LIN {X 0,Y 179.532,Z 337.35,A -85,B 0,C 180,E1 -23453.668,E2 -23453.668} C_VEL
LIN {X 0,Y 179.263,Z 347.509,A -85,B 0,C 180,E1 -23456.334,E2 -23456.334} C_VEL
LIN {X 0,Y 178.405,Z 355.039,A -85,B 0,C 180,E1 -23458.536,E2 -23458.536} C_VEL
LIN {X 0,Y 174.902,Z 363.864,A -85,B 0,C 180,E1 -23461.171,E2 -23461.171} C_VEL
LIN {X 0,Y 171.795,Z 371.251,A -85,B 0,C 180,E1 -23463.957,E2 -23463.957} C_VEL
LIN {X 0,Y 168.803,Z 378.338,A -85,B 0,C 180,E1 -23467.349,E2 -23467.349} C_VEL
LIN {X 0,Y 166.619,Z 383.189,A -85,B 0,C 180,E1 -23470.279,E2 -23470.279} C_VEL
LIN {X 0,Y 164.438,Z 387.902,A -85,B 0,C 180,E1 -23473.87,E2 -23473.87} C_VEL
LIN {X 0,Y 163.052,Z 391.511,A -85,B 0,C 180,E1 -23477.554,E2 -23477.554} C_VEL
LIN {X 0,Y 162.401,Z 393.372,A -85,B 0,C 180,E1 -23480.031,E2 -23480.031} C_VEL
LIN {X 0,Y 161.998,Z 394.77,A -85,B 0,C 180,E1 -23482.521,E2 -23482.521} C_VEL
LIN {X 0,Y 161.792,Z 395.77,A -85,B 0,C 180,E1 -23485.016,E2 -23485.016} C_VEL
LIN {X 0,Y 161.766,Z 396.433,A -85,B 0,C 180,E1 -23487.777,E2 -23487.777} C_VEL
LIN {X 0,Y 161.898,Z 396.597,A -85,B 0,C 180,E1 -23490,E2 -23490} C_VEL
LIN {X 0,Y 161.765,Z 396.367,A -85,B 0,C 180,E1 -23492.49,E2 -23492.49} C_VEL
LIN {X 0,Y 161.973,Z 394.738,A -85,B 0,C 180,E1 -23497.479,E2 -23497.479} C_VEL
LIN {X 0,Y 162.397,Z 393.327,A -85,B 0,C 180,E1 -23499.968,E2 -23499.968} C_VEL
LIN {X 0,Y 163.451,Z 390.371,A -85,B 0,C 180,E1 -23503.679,E2 -23503.679} C_VEL
LIN {X 0,Y 165.064,Z 386.378,A -85,B 0,C 180,E1 -23507.34,E2 -23507.34} C_VEL
LIN {X 0,Y 167.85,Z 380.247,A -85,B 0,C 180,E1 -23511.492,E2 -23511.492} C_VEL
LIN {X 0,Y 171.05,Z 373.162,A -85,B 0,C 180,E1 -23515.115,E2 -23515.115} C_VEL
LIN {X 0,Y 174.277,Z 365.256,A -85,B 0,C 180,E1 -23518.284,E2 -23518.284} C_VEL
LIN {X 0,Y 176.008,Z 361.044,A -85,B 0,C 180,E1 -23519.667,E2 -23519.667} C_VEL
LIN {X 0,Y 176.715,Z 358.334,A -85,B 0,C 180,E1 -23520.56,E2 -23520.56} C_VEL
LIN {X 0,Y 176.609,Z 354.361,A -85,B 0,C 180,E1 -23521.984,E2 -23521.984} C_VEL
LIN {X 0,Y 175.665,Z 350.503,A -85,B 0,C 180,E1 -23523.438,E2 -23523.438} C_VEL
LIN {X 0,Y 173.47,Z 342.313,A -85,B 0,C 180,E1 -23526.334,E2 -23526.334} C_VEL
LIN {X 0,Y 173.279,Z 339.26,A -85,B 0,C 180,E1 -23527.216,E2 -23527.216} C_VEL
LIN {X 0,Y 172.896,Z 328.815,A -85,B 0,C 180,E1 -23529.893,E2 -23529.893} C_VEL
LIN {X 0,Y 171.766,Z 319.398,A -85,B 0,C 180,E1 -23532.155,E2 -23532.155} C_VEL
LIN {X 0,Y 170.094,Z 313.723,A -85,B 0,C 180,E1 -23533.691,E2 -23533.691} C_VEL
LIN {X 0,Y 165.868,Z 303.988,A -85,B 0,C 180,E1 -23536.632,E2 -23536.632} C_VEL
LIN {X 0,Y 163.409,Z 299.193,A -85,B 0,C 180,E1 -23538.192,E2 -23538.192} C_VEL
LIN {X 0,Y 161.486,Z 295.384,A -85,B 0,C 180,E1 -23539.427,E2 -23539.427} C_VEL
LIN {X 0,Y 158.662,Z 290.982,A -85,B 0,C 180,E1 -23541.1,E2 -23541.1} C_VEL
LIN {X 0,Y 158.114,Z 289.125,A -85,B 0,C 180,E1 -23541.578,E2 -23541.578} C_VEL
LIN {X 0,Y 157.959,Z 287.633,A -85,B 0,C 180,E1 -23544.662,E2 -23544.662} C_VEL
LIN {X 0,Y 157.689,Z 286.213,A -85,B 0,C 180,E1 -23547.866,E2 -23547.866} C_VEL
LIN {X 0,Y 157.309,Z 283.978,A -85,B 0,C 180,E1 -23553.464,E2 -23553.464} C_VEL
LIN {X 0,Y 157.392,Z 283.88,A -85,B 0,C 180,E1 -23559.67,E2 -23559.67} C_VEL
LIN {X 0,Y 157.454,Z 283.87,A -85,B 0,C 180,E1 -23564.466,E2 -23564.466} C_VEL
LIN {X 0,Y 157.69,Z 283.841,A -85,B 0,C 180,E1 -23569.731,E2 -23569.731} C_VEL
LIN {X 0,Y 157.767,Z 283.83,A -85,B 0,C 180,E1 -23572.32,E2 -23572.32} C_VEL
LIN {X 0,Y 158.249,Z 283.773,A -85,B 0,C 180,E1 -23580,E2 -23580} C_VEL
LIN {X 0,Y 157.764,Z 283.832,A -85,B 0,C 180,E1 -23587.68,E2 -23587.68} C_VEL
LIN {X 0,Y 157.634,Z 283.847,A -85,B 0,C 180,E1 -23591.23,E2 -23591.23} C_VEL
LIN {X 0,Y 157.436,Z 283.871,A -85,B 0,C 180,E1 -23595.536,E2 -23595.536} C_VEL
LIN {X 0,Y 157.367,Z 283.88,A -85,B 0,C 180,E1 -23600.933,E2 -23600.933} C_VEL
LIN {X 0,Y 157.31,Z 283.888,A -85,B 0,C 180,E1 -23606.681,E2 -23606.681} C_VEL
LIN {X 0,Y 157.279,Z 283.895,A -85,B 0,C 180,E1 -23612.427,E2 -23612.427} C_VEL
LIN {X 0,Y 157.233,Z 283.899,A -85,B 0,C 180,E1 -23617.483,E2 -23617.483} C_VEL
LIN {X 0,Y 157.261,Z 284.165,A -85,B 0,C 180,E1 -23618.179,E2 -23618.179} C_VEL
LIN {X 0,Y 158.285,Z 286.868,A -85,B 0,C 180,E1 -23618.941,E2 -23618.941} C_VEL
LIN {X 0,Y 160.69,Z 289.727,A -85,B 0,C 180,E1 -23620.31,E2 -23620.31} C_VEL
LIN {X 0,Y 162.703,Z 293.411,A -85,B 0,C 180,E1 -23621.616,E2 -23621.616} C_VEL
LIN {X 0,Y 163.922,Z 295.532,A -85,B 0,C 180,E1 -23622.371,E2 -23622.371} C_VEL
LIN {X 0,Y 166.248,Z 299.878,A -85,B 0,C 180,E1 -23623.888,E2 -23623.888} C_VEL
LIN {X 0,Y 170.184,Z 308.553,A -85,B 0,C 180,E1 -23626.703,E2 -23626.703} C_VEL
LIN {X 0,Y 173.03,Z 318.057,A -85,B 0,C 180,E1 -23629.468,E2 -23629.468} C_VEL
LIN {X 0,Y 174.681,Z 328.982,A -85,B 0,C 180,E1 -23632.527,E2 -23632.527} C_VEL
LIN {X 0,Y 175.059,Z 338.675,A -85,B 0,C 180,E1 -23635.374,E2 -23635.374} C_VEL
LIN {X 0,Y 174.874,Z 343.244,A -85,B 0,C 180,E1 -23636.799,E2 -23636.799} C_VEL
LIN {X 0,Y 171.561,Z 351.776,A -85,B 0,C 180,E1 -23639.2,E2 -23639.2} C_VEL
LIN {X 0,Y 168.32,Z 359.639,A -85,B 0,C 180,E1 -23641.99,E2 -23641.99} C_VEL
LIN {X 0,Y 164.672,Z 367.301,A -85,B 0,C 180,E1 -23645.41,E2 -23645.41} C_VEL
LIN {X 0,Y 161.071,Z 374.352,A -85,B 0,C 180,E1 -23649.57,E2 -23649.57} C_VEL
LIN {X 0,Y 158.731,Z 379.04,A -85,B 0,C 180,E1 -23653.274,E2 -23653.274} C_VEL
LIN {X 0,Y 156.993,Z 382.624,A -85,B 0,C 180,E1 -23657.066,E2 -23657.066} C_VEL
LIN {X 0,Y 156.094,Z 384.475,A -85,B 0,C 180,E1 -23659.625,E2 -23659.625} C_VEL
LIN {X 0,Y 155.506,Z 385.863,A -85,B 0,C 180,E1 -23662.208,E2 -23662.208} C_VEL
LIN {X 0,Y 154.905,Z 387.455,A -85,B 0,C 180,E1 -23667.4,E2 -23667.4} C_VEL
LIN {X 0,Y 154.86,Z 387.681,A -85,B 0,C 180,E1 -23670,E2 -23670} C_VEL
LIN {X 0,Y 154.952,Z 387.273,A -85,B 0,C 180,E1 -23673.771,E2 -23673.771} C_VEL
LIN {X 0,Y 155.507,Z 385.933,A -85,B 0,C 180,E1 -23677.793,E2 -23677.793} C_VEL
LIN {X 0,Y 156.093,Z 384.576,A -85,B 0,C 180,E1 -23680.376,E2 -23680.376} C_VEL
LIN {X 0,Y 157.48,Z 381.707,A -85,B 0,C 180,E1 -23684.209,E2 -23684.209} C_VEL
LIN {X 0,Y 159.422,Z 377.814,A -85,B 0,C 180,E1 -23687.975,E2 -23687.975} C_VEL
LIN {X 0,Y 161.963,Z 372.79,A -85,B 0,C 180,E1 -23691.644,E2 -23691.644} C_VEL
LIN {X 0,Y 165.148,Z 366.457,A -85,B 0,C 180,E1 -23695.186,E2 -23695.186} C_VEL
LIN {X 0,Y 168.761,Z 358.637,A -85,B 0,C 180,E1 -23698.569,E2 -23698.569} C_VEL
LIN {X 0,Y 172.052,Z 350.641,A -85,B 0,C 180,E1 -23701.319,E2 -23701.319} C_VEL
LIN {X 0,Y 174.992,Z 342.742,A -85,B 0,C 180,E1 -23703.52,E2 -23703.52} C_VEL
LIN {X 0,Y 175.049,Z 333.244,A -85,B 0,C 180,E1 -23706.41,E2 -23706.41} C_VEL
LIN {X 0,Y 174.114,Z 324.129,A -85,B 0,C 180,E1 -23709.032,E2 -23709.032} C_VEL
LIN {X 0,Y 172.377,Z 315.457,A -85,B 0,C 180,E1 -23711.48,E2 -23711.48} C_VEL
LIN {X 0,Y 169.606,Z 307.081,A -85,B 0,C 180,E1 -23713.964,E2 -23713.964} C_VEL
LIN {X 0,Y 165.424,Z 298.191,A -85,B 0,C 180,E1 -23716.883,E2 -23716.883} C_VEL
LIN {X 0,Y 162.733,Z 293.422,A -85,B 0,C 180,E1 -23718.6,E2 -23718.6} C_VEL
LIN {X 0,Y 160.797,Z 289.973,A -85,B 0,C 180,E1 -23719.852,E2 -23719.852} C_VEL
LIN {X 0,Y 159.998,Z 288.814,A -85,B 0,C 180,E1 -23720.324,E2 -23720.324} C_VEL
LIN {X 0,Y 157.92,Z 286.258,A -85,B 0,C 180,E1 -23721.539,E2 -23721.539} C_VEL
LIN {X 0,Y 157.234,Z 283.938,A -85,B 0,C 180,E1 -23722.205,E2 -23722.205} C_VEL
LIN {X 0,Y 157.293,Z 283.894,A -85,B 0,C 180,E1 -23724.489,E2 -23724.489} C_VEL
LIN {X 0,Y 157.297,Z 283.889,A -85,B 0,C 180,E1 -23728.095,E2 -23728.095} C_VEL
LIN {X 0,Y 157.317,Z 283.885,A -85,B 0,C 180,E1 -23733.465,E2 -23733.465} C_VEL
LIN {X 0,Y 157.394,Z 283.878,A -85,B 0,C 180,E1 -23739.67,E2 -23739.67} C_VEL
LIN {X 0,Y 157.439,Z 283.874,A -85,B 0,C 180,E1 -23744.464,E2 -23744.464} C_VEL
LIN {X 0,Y 157.691,Z 283.842,A -85,B 0,C 180,E1 -23749.731,E2 -23749.731} C_VEL
LIN {X 0,Y 157.765,Z 283.834,A -85,B 0,C 180,E1 -23752.32,E2 -23752.32} C_VEL
LIN {X 0,Y 158.24,Z 283.773,A -85,B 0,C 180,E1 -23760,E2 -23760} C_VEL
LIN {X 0,Y 157.714,Z 283.838,A -85,B 0,C 180,E1 -23765.113,E2 -23765.113} C_VEL
LIN {X 0,Y 157.769,Z 283.83,A -85,B 0,C 180,E1 -23767.68,E2 -23767.68} C_VEL
LIN {X 0,Y 157.639,Z 283.849,A -85,B 0,C 180,E1 -23771.237,E2 -23771.237} C_VEL
LIN {X 0,Y 157.444,Z 283.872,A -85,B 0,C 180,E1 -23775.535,E2 -23775.535} C_VEL
LIN {X 0,Y 157.369,Z 283.882,A -85,B 0,C 180,E1 -23780.933,E2 -23780.933} C_VEL
LIN {X 0,Y 157.322,Z 284.102,A -85,B 0,C 180,E1 -23786.688,E2 -23786.688} C_VEL
LIN {X 0,Y 157.722,Z 286.361,A -85,B 0,C 180,E1 -23792.324,E2 -23792.324} C_VEL
LIN {X 0,Y 158.069,Z 288.406,A -85,B 0,C 180,E1 -23796.84,E2 -23796.84} C_VEL
LIN {X 0,Y 158.146,Z 289.255,A -85,B 0,C 180,E1 -23798.351,E2 -23798.351} C_VEL
LIN {X 0,Y 159.201,Z 292.065,A -85,B 0,C 180,E1 -23799.106,E2 -23799.106} C_VEL
LIN {X 0,Y 161.514,Z 295.42,A -85,B 0,C 180,E1 -23800.447,E2 -23800.447} C_VEL
LIN {X 0,Y 163.571,Z 299.367,A -85,B 0,C 180,E1 -23801.757,E2 -23801.757} C_VEL
LIN {X 0,Y 167.057,Z 306.433,A -85,B 0,C 180,E1 -23804.012,E2 -23804.012} C_VEL
LIN {X 0,Y 170.194,Z 313.991,A -85,B 0,C 180,E1 -23806.273,E2 -23806.273} C_VEL
LIN {X 0,Y 171.979,Z 320.43,A -85,B 0,C 180,E1 -23808.002,E2 -23808.002} C_VEL
LIN {X 0,Y 173.096,Z 330.614,A -85,B 0,C 180,E1 -23810.483,E2 -23810.483} C_VEL
LIN {X 0,Y 173.321,Z 341.13,A -85,B 0,C 180,E1 -23813.217,E2 -23813.217} C_VEL
LIN {X 0,Y 172.668,Z 350.737,A -85,B 0,C 180,E1 -23815.967,E2 -23815.967} C_VEL
LIN {X 0,Y 172.155,Z 354.834,A -85,B 0,C 180,E1 -23817.254,E2 -23817.254} C_VEL
LIN {X 0,Y 170.919,Z 358.58,A -85,B 0,C 180,E1 -23818.381,E2 -23818.381} C_VEL
LIN {X 0,Y 166.674,Z 368.22,A -85,B 0,C 180,E1 -23821.681,E2 -23821.681} C_VEL
LIN {X 0,Y 163.351,Z 375.904,A -85,B 0,C 180,E1 -23825.198,E2 -23825.198} C_VEL
LIN {X 0,Y 160.81,Z 381.168,A -85,B 0,C 180,E1 -23828.193,E2 -23828.193} C_VEL
LIN {X 0,Y 158.291,Z 386.268,A -85,B 0,C 180,E1 -23831.893,E2 -23831.893} C_VEL
LIN {X 0,Y 156.526,Z 390.236,A -85,B 0,C 180,E1 -23835.703,E2 -23835.703} C_VEL
LIN {X 0,Y 155.402,Z 393.173,A -85,B 0,C 180,E1 -23839.578,E2 -23839.578} C_VEL
LIN {X 0,Y 154.948,Z 394.57,A -85,B 0,C 180,E1 -23842.179,E2 -23842.179} C_VEL
LIN {X 0,Y 154.712,Z 395.57,A -85,B 0,C 180,E1 -23844.787,E2 -23844.787} C_VEL
LIN {X 0,Y 154.684,Z 396.297,A -85,B 0,C 180,E1 -23848.304,E2 -23848.304} C_VEL
LIN {X 0,Y 154.796,Z 396.397,A -85,B 0,C 180,E1 -23850,E2 -23850} C_VEL
LIN {X 0,Y 154.666,Z 396.167,A -85,B 0,C 180,E1 -23852.604,E2 -23852.604} C_VEL
LIN {X 0,Y 154.695,Z 395.547,A -85,B 0,C 180,E1 -23855.213,E2 -23855.213} C_VEL
LIN {X 0,Y 154.929,Z 394.538,A -85,B 0,C 180,E1 -23857.821,E2 -23857.821} C_VEL
LIN {X 0,Y 155.399,Z 393.126,A -85,B 0,C 180,E1 -23860.422,E2 -23860.422} C_VEL
LIN {X 0,Y 156.525,Z 390.17,A -85,B 0,C 180,E1 -23864.297,E2 -23864.297} C_VEL
LIN {X 0,Y 158.289,Z 386.177,A -85,B 0,C 180,E1 -23868.107,E2 -23868.107} C_VEL
LIN {X 0,Y 161.222,Z 380.045,A -85,B 0,C 180,E1 -23872.422,E2 -23872.422} C_VEL
LIN {X 0,Y 164.353,Z 373.538,A -85,B 0,C 180,E1 -23875.895,E2 -23875.895} C_VEL
LIN {X 0,Y 168.039,Z 365.054,A -85,B 0,C 180,E1 -23879.434,E2 -23879.434} C_VEL
LIN {X 0,Y 171.625,Z 356.544,A -85,B 0,C 180,E1 -23882.164,E2 -23882.164} C_VEL
LIN {X 0,Y 172.9,Z 348.293,A -85,B 0,C 180,E1 -23884.685,E2 -23884.685} C_VEL
LIN {X 0,Y 173.279,Z 339.26,A -85,B 0,C 180,E1 -23887.216,E2 -23887.216} C_VEL
LIN {X 0,Y 172.779,Z 334.847,A -85,B 0,C 180,E1 -23888.508,E2 -23888.508} C_VEL
LIN {X 0,Y 171.404,Z 330.8,A -85,B 0,C 180,E1 -23889.883,E2 -23889.883} C_VEL
LIN {X 0,Y 167.438,Z 323.176,A -85,B 0,C 180,E1 -23892.745,E2 -23892.745} C_VEL
LIN {X 0,Y 164.93,Z 317.767,A -85,B 0,C 180,E1 -23894.624,E2 -23894.624} C_VEL
LIN {X 0,Y 161.37,Z 308.826,A -85,B 0,C 180,E1 -23897.543,E2 -23897.543} C_VEL
LIN {X 0,Y 159.078,Z 304.056,A -85,B 0,C 180,E1 -23899.23,E2 -23899.23} C_VEL
LIN {X 0,Y 156.751,Z 299.454,A -85,B 0,C 180,E1 -23900.913,E2 -23900.913} C_VEL
LIN {X 0,Y 154.665,Z 295.601,A -85,B 0,C 180,E1 -23902.408,E2 -23902.408} C_VEL
LIN {X 0,Y 153.755,Z 294.127,A -85,B 0,C 180,E1 -23903.022,E2 -23903.022} C_VEL
LIN {X 0,Y 151.625,Z 290.908,A -85,B 0,C 180,E1 -23904.49,E2 -23904.49} C_VEL
LIN {X 0,Y 150.932,Z 288.787,A -85,B 0,C 180,E1 -23905.221,E2 -23905.221} C_VEL
LIN {X 0,Y 150.611,Z 287.176,A -85,B 0,C 180,E1 -23909.116,E2 -23909.116} C_VEL
LIN {X 0,Y 150.245,Z 284.971,A -85,B 0,C 180,E1 -23915.103,E2 -23915.103} C_VEL
LIN {X 0,Y 150.36,Z 284.757,A -85,B 0,C 180,E1 -23920.902,E2 -23920.902} C_VEL
LIN {X 0,Y 150.436,Z 284.743,A -85,B 0,C 180,E1 -23926.492,E2 -23926.492} C_VEL
LIN {X 0,Y 150.612,Z 284.721,A -85,B 0,C 180,E1 -23929.243,E2 -23929.243} C_VEL
LIN {X 0,Y 150.705,Z 284.709,A -85,B 0,C 180,E1 -23931.958,E2 -23931.958} C_VEL
LIN {X 0,Y 151.21,Z 284.65,A -85,B 0,C 180,E1 -23940,E2 -23940} C_VEL
LIN {X 0,Y 150.702,Z 284.71,A -85,B 0,C 180,E1 -23948.043,E2 -23948.043} C_VEL
LIN {X 0,Y 150.576,Z 284.725,A -85,B 0,C 180,E1 -23951.433,E2 -23951.433} C_VEL
LIN {X 0,Y 150.348,Z 284.756,A -85,B 0,C 180,E1 -23956.288,E2 -23956.288} C_VEL
LIN {X 0,Y 150.35,Z 284.755,A -85,B 0,C 180,E1 -23960.79,E2 -23960.79} C_VEL
LIN {X 0,Y 150.242,Z 284.769,A -85,B 0,C 180,E1 -23967.28,E2 -23967.28} C_VEL
LIN {X 0,Y 150.22,Z 284.774,A -85,B 0,C 180,E1 -23972.635,E2 -23972.635} C_VEL
LIN {X 0,Y 150.222,Z 284.912,A -85,B 0,C 180,E1 -23974.661,E2 -23974.661} C_VEL
LIN {X 0,Y 151.197,Z 287.513,A -85,B 0,C 180,E1 -23975.523,E2 -23975.523} C_VEL
LIN {X 0,Y 153.217,Z 289.733,A -85,B 0,C 180,E1 -23976.851,E2 -23976.851} C_VEL
LIN {X 0,Y 153.8,Z 290.482,A -85,B 0,C 180,E1 -23977.238,E2 -23977.238} C_VEL
LIN {X 0,Y 155.531,Z 293.516,A -85,B 0,C 180,E1 -23978.515,E2 -23978.515} C_VEL
LIN {X 0,Y 156.846,Z 295.277,A -85,B 0,C 180,E1 -23979.37,E2 -23979.37} C_VEL
LIN {X 0,Y 160.981,Z 303.073,A -85,B 0,C 180,E1 -23982.416,E2 -23982.416} C_VEL
LIN {X 0,Y 164.907,Z 312.263,A -85,B 0,C 180,E1 -23985.645,E2 -23985.645} C_VEL
LIN {X 0,Y 167.208,Z 320.482,A -85,B 0,C 180,E1 -23988.251,E2 -23988.251} C_VEL
LIN {X 0,Y 168.57,Z 330.571,A -85,B 0,C 180,E1 -23991.29,E2 -23991.29} C_VEL
LIN {X 0,Y 168.827,Z 339.162,A -85,B 0,C 180,E1 -23993.986,E2 -23993.986} C_VEL
LIN {X 0,Y 168.583,Z 344.502,A -85,B 0,C 180,E1 -23995.751,E2 -23995.751} C_VEL
LIN {X 0,Y 164.42,Z 354.389,A -85,B 0,C 180,E1 -23998.747,E2 -23998.747} C_VEL
LIN {X 0,Y 160.74,Z 362.559,A -85,B 0,C 180,E1 -24001.965,E2 -24001.965} C_VEL
LIN {X 0,Y 157.061,Z 369.724,A -85,B 0,C 180,E1 -24005.549,E2 -24005.549} C_VEL
LIN {X 0,Y 154.424,Z 374.553,A -85,B 0,C 180,E1 -24008.649,E2 -24008.649} C_VEL
LIN {X 0,Y 151.952,Z 379.241,A -85,B 0,C 180,E1 -24012.505,E2 -24012.505} C_VEL
LIN {X 0,Y 150.067,Z 382.825,A -85,B 0,C 180,E1 -24016.458,E2 -24016.458} C_VEL
LIN {X 0,Y 149.122,Z 384.675,A -85,B 0,C 180,E1 -24019.134,E2 -24019.134} C_VEL
LIN {X 0,Y 148.47,Z 386.063,A -85,B 0,C 180,E1 -24021.836,E2 -24021.836} C_VEL
LIN {X 0,Y 147.84,Z 387.549,A -85,B 0,C 180,E1 -24026.662,E2 -24026.662} C_VEL
LIN {X 0,Y 147.766,Z 387.881,A -85,B 0,C 180,E1 -24030,E2 -24030} C_VEL
LIN {X 0,Y 147.84,Z 387.579,A -85,B 0,C 180,E1 -24033.338,E2 -24033.338} C_VEL
LIN {X 0,Y 148.47,Z 386.133,A -85,B 0,C 180,E1 -24038.164,E2 -24038.164} C_VEL
LIN {X 0,Y 149.121,Z 384.775,A -85,B 0,C 180,E1 -24040.867,E2 -24040.867} C_VEL
LIN {X 0,Y 150.6,Z 381.906,A -85,B 0,C 180,E1 -24044.873,E2 -24044.873} C_VEL
LIN {X 0,Y 152.692,Z 378.012,A -85,B 0,C 180,E1 -24048.796,E2 -24048.796} C_VEL
LIN {X 0,Y 155.393,Z 372.988,A -85,B 0,C 180,E1 -24052.609,E2 -24052.609} C_VEL
LIN {X 0,Y 158.762,Z 366.655,A -85,B 0,C 180,E1 -24056.275,E2 -24056.275} C_VEL
LIN {X 0,Y 162.445,Z 359.077,A -85,B 0,C 180,E1 -24059.672,E2 -24059.672} C_VEL
LIN {X 0,Y 166.017,Z 350.839,A -85,B 0,C 180,E1 -24062.595,E2 -24062.595} C_VEL
LIN {X 0,Y 168.709,Z 344.004,A -85,B 0,C 180,E1 -24064.582,E2 -24064.582} C_VEL
LIN {X 0,Y 168.898,Z 334.156,A -85,B 0,C 180,E1 -24067.757,E2 -24067.757} C_VEL
LIN {X 0,Y 168.019,Z 325.162,A -85,B 0,C 180,E1 -24070.531,E2 -24070.531} C_VEL
LIN {X 0,Y 166.307,Z 316.8,A -85,B 0,C 180,E1 -24073.11,E2 -24073.11} C_VEL
LIN {X 0,Y 164.031,Z 309.92,A -85,B 0,C 180,E1 -24075.358,E2 -24075.358} C_VEL
LIN {X 0,Y 160.626,Z 302.512,A -85,B 0,C 180,E1 -24078.058,E2 -24078.058} C_VEL
LIN {X 0,Y 158.253,Z 298.012,A -85,B 0,C 180,E1 -24079.809,E2 -24079.809} C_VEL
LIN {X 0,Y 156.268,Z 294.386,A -85,B 0,C 180,E1 -24081.267,E2 -24081.267} C_VEL
LIN {X 0,Y 154.194,Z 291.412,A -85,B 0,C 180,E1 -24082.69,E2 -24082.69} C_VEL
LIN {X 0,Y 153.522,Z 289.91,A -85,B 0,C 180,E1 -24083.235,E2 -24083.235} C_VEL
LIN {X 0,Y 151.261,Z 287.635,A -85,B 0,C 180,E1 -24084.698,E2 -24084.698} C_VEL
LIN {X 0,Y 150.27,Z 285.206,A -85,B 0,C 180,E1 -24085.555,E2 -24085.555} C_VEL
LIN {X 0,Y 150.19,Z 284.773,A -85,B 0,C 180,E1 -24085.737,E2 -24085.737} C_VEL
LIN {X 0,Y 150.21,Z 284.769,A -85,B 0,C 180,E1 -24089.025,E2 -24089.025} C_VEL
LIN {X 0,Y 150.243,Z 284.763,A -85,B 0,C 180,E1 -24092.72,E2 -24092.72} C_VEL
LIN {X 0,Y 150.351,Z 284.757,A -85,B 0,C 180,E1 -24099.21,E2 -24099.21} C_VEL
LIN {X 0,Y 150.351,Z 284.758,A -85,B 0,C 180,E1 -24103.712,E2 -24103.712} C_VEL
LIN {X 0,Y 150.611,Z 284.725,A -85,B 0,C 180,E1 -24109.242,E2 -24109.242} C_VEL
LIN {X 0,Y 150.703,Z 284.713,A -85,B 0,C 180,E1 -24111.958,E2 -24111.958} C_VEL
LIN {X 0,Y 151.201,Z 284.65,A -85,B 0,C 180,E1 -24120,E2 -24120} C_VEL
LIN {X 0,Y 150.706,Z 284.711,A -85,B 0,C 180,E1 -24128.042,E2 -24128.042} C_VEL
LIN {X 0,Y 150.579,Z 284.729,A -85,B 0,C 180,E1 -24131.438,E2 -24131.438} C_VEL
LIN {X 0,Y 150.356,Z 284.757,A -85,B 0,C 180,E1 -24136.287,E2 -24136.287} C_VEL
LIN {X 0,Y 150.351,Z 284.757,A -85,B 0,C 180,E1 -24140.79,E2 -24140.79} C_VEL
LIN {X 0,Y 150.25,Z 285.039,A -85,B 0,C 180,E1 -24144.896,E2 -24144.896} C_VEL
LIN {X 0,Y 150.435,Z 286.08,A -85,B 0,C 180,E1 -24147.851,E2 -24147.851} C_VEL
LIN {X 0,Y 150.808,Z 288.09,A -85,B 0,C 180,E1 -24152.981,E2 -24152.981} C_VEL
LIN {X 0,Y 150.969,Z 288.997,A -85,B 0,C 180,E1 -24154.769,E2 -24154.769} C_VEL
LIN {X 0,Y 152.29,Z 292.195,A -85,B 0,C 180,E1 -24155.839,E2 -24155.839} C_VEL
LIN {X 0,Y 154.539,Z 295.267,A -85,B 0,C 180,E1 -24157.328,E2 -24157.328} C_VEL
LIN {X 0,Y 156.587,Z 299.181,A -85,B 0,C 180,E1 -24158.823,E2 -24158.823} C_VEL
LIN {X 0,Y 157.546,Z 300.81,A -85,B 0,C 180,E1 -24159.471,E2 -24159.471} C_VEL
LIN {X 0,Y 160.328,Z 306.492,A -85,B 0,C 180,E1 -24161.513,E2 -24161.513} C_VEL
LIN {X 0,Y 164.171,Z 315.549,A -85,B 0,C 180,E1 -24164.571,E2 -24164.571} C_VEL
LIN {X 0,Y 166.351,Z 322.936,A -85,B 0,C 180,E1 -24166.795,E2 -24166.795} C_VEL
LIN {X 0,Y 167.216,Z 333.484,A -85,B 0,C 180,E1 -24169.568,E2 -24169.568} C_VEL
LIN {X 0,Y 167.12,Z 343.551,A -85,B 0,C 180,E1 -24172.39,E2 -24172.39} C_VEL
LIN {X 0,Y 166.22,Z 352.654,A -85,B 0,C 180,E1 -24175.194,E2 -24175.194} C_VEL
LIN {X 0,Y 165.557,Z 356.585,A -85,B 0,C 180,E1 -24176.505,E2 -24176.505} C_VEL
LIN {X 0,Y 161.85,Z 365.045,A -85,B 0,C 180,E1 -24179.321,E2 -24179.321} C_VEL
LIN {X 0,Y 157.893,Z 373.389,A -85,B 0,C 180,E1 -24182.901,E2 -24182.901} C_VEL
LIN {X 0,Y 155.208,Z 378.961,A -85,B 0,C 180,E1 -24185.95,E2 -24185.95} C_VEL
LIN {X 0,Y 152.366,Z 384.481,A -85,B 0,C 180,E1 -24189.76,E2 -24189.76} C_VEL
LIN {X 0,Y 150.135,Z 388.812,A -85,B 0,C 180,E1 -24193.688,E2 -24193.688} C_VEL
LIN {X 0,Y 149.136,Z 391.111,A -85,B 0,C 180,E1 -24196.371,E2 -24196.371} C_VEL
LIN {X 0,Y 148.388,Z 392.973,A -85,B 0,C 180,E1 -24199.079,E2 -24199.079} C_VEL
LIN {X 0,Y 147.897,Z 394.37,A -85,B 0,C 180,E1 -24201.804,E2 -24201.804} C_VEL
LIN {X 0,Y 147.634,Z 395.37,A -85,B 0,C 180,E1 -24204.536,E2 -24204.536} C_VEL
LIN {X 0,Y 147.622,Z 396.131,A -85,B 0,C 180,E1 -24208.772,E2 -24208.772} C_VEL
LIN {X 0,Y 147.63,Z 396.118,A -85,B 0,C 180,E1 -24211.362,E2 -24211.362} C_VEL
LIN {X 0,Y 147.622,Z 395.346,A -85,B 0,C 180,E1 -24215.463,E2 -24215.463} C_VEL
LIN {X 0,Y 147.883,Z 394.337,A -85,B 0,C 180,E1 -24218.196,E2 -24218.196} C_VEL
LIN {X 0,Y 148.386,Z 392.925,A -85,B 0,C 180,E1 -24220.921,E2 -24220.921} C_VEL
LIN {X 0,Y 149.625,Z 389.968,A -85,B 0,C 180,E1 -24224.971,E2 -24224.971} C_VEL
LIN {X 0,Y 151.545,Z 385.975,A -85,B 0,C 180,E1 -24228.943,E2 -24228.943} C_VEL
LIN {X 0,Y 154.656,Z 379.843,A -85,B 0,C 180,E1 -24233.43,E2 -24233.43} C_VEL
LIN {X 0,Y 157.473,Z 374.39,A -85,B 0,C 180,E1 -24236.506,E2 -24236.506} C_VEL
LIN {X 0,Y 161.165,Z 366.342,A -85,B 0,C 180,E1 -24240.098,E2 -24240.098} C_VEL
LIN {X 0,Y 164.876,Z 358.148,A -85,B 0,C 180,E1 -24242.921,E2 -24242.921} C_VEL
LIN {X 0,Y 165.84,Z 354.367,A -85,B 0,C 180,E1 -24244.16,E2 -24244.16} C_VEL
LIN {X 0,Y 166.814,Z 346.89,A -85,B 0,C 180,E1 -24246.527,E2 -24246.527} C_VEL
LIN {X 0,Y 167.173,Z 336.191,A -85,B 0,C 180,E1 -24249.606,E2 -24249.606} C_VEL
LIN {X 0,Y 166.542,Z 325.417,A -85,B 0,C 180,E1 -24252.469,E2 -24252.469} C_VEL
LIN {X 0,Y 165.681,Z 320.289,A -85,B 0,C 180,E1 -24253.853,E2 -24253.853} C_VEL
LIN {X 0,Y 164.93,Z 317.767,A -85,B 0,C 180,E1 -24254.624,E2 -24254.624} C_VEL
LIN {X 0,Y 163.441,Z 315.395,A -85,B 0,C 180,E1 -24255.592,E2 -24255.592} C_VEL
LIN {X 0,Y 159.904,Z 312.847,A -85,B 0,C 180,E1 -24257.382,E2 -24257.382} C_VEL
LIN {X 0,Y 155.582,Z 309.957,A -85,B 0,C 180,E1 -24259.664,E2 -24259.664} C_VEL
LIN {X 0,Y 154.497,Z 308.525,A -85,B 0,C 180,E1 -24260.407,E2 -24260.407} C_VEL
LIN {X 0,Y 152.646,Z 304.534,A -85,B 0,C 180,E1 -24261.98,E2 -24261.98} C_VEL
LIN {X 0,Y 150.102,Z 299.628,A -85,B 0,C 180,E1 -24264.075,E2 -24264.075} C_VEL
LIN {X 0,Y 147.995,Z 295.975,A -85,B 0,C 180,E1 -24265.792,E2 -24265.792} C_VEL
LIN {X 0,Y 147.259,Z 294.473,A -85,B 0,C 180,E1 -24266.431,E2 -24266.431} C_VEL
LIN {X 0,Y 144.698,Z 291.323,A -85,B 0,C 180,E1 -24268.423,E2 -24268.423} C_VEL
LIN {X 0,Y 143.616,Z 288.48,A -85,B 0,C 180,E1 -24269.59,E2 -24269.59} C_VEL
LIN {X 0,Y 143.355,Z 286.976,A -85,B 0,C 180,E1 -24273.818,E2 -24273.818} C_VEL
LIN {X 0,Y 143.275,Z 285.64,A -85,B 0,C 180,E1 -24278.748,E2 -24278.748} C_VEL
LIN {X 0,Y 143.302,Z 285.635,A -85,B 0,C 180,E1 -24282.887,E2 -24282.887} C_VEL
LIN {X 0,Y 143.538,Z 285.603,A -85,B 0,C 180,E1 -24288.706,E2 -24288.706} C_VEL
LIN {X 0,Y 143.626,Z 285.592,A -85,B 0,C 180,E1 -24291.559,E2 -24291.559} C_VEL
LIN {X 0,Y 144.168,Z 285.527,A -85,B 0,C 180,E1 -24300,E2 -24300} C_VEL
LIN {X 0,Y 143.624,Z 285.591,A -85,B 0,C 180,E1 -24308.442,E2 -24308.442} C_VEL
LIN {X 0,Y 143.502,Z 285.606,A -85,B 0,C 180,E1 -24311.623,E2 -24311.623} C_VEL
LIN {X 0,Y 143.292,Z 285.636,A -85,B 0,C 180,E1 -24317.115,E2 -24317.115} C_VEL
LIN {X 0,Y 143.275,Z 285.635,A -85,B 0,C 180,E1 -24321.252,E2 -24321.252} C_VEL
LIN {X 0,Y 143.189,Z 285.65,A -85,B 0,C 180,E1 -24327.936,E2 -24327.936} C_VEL
LIN {X 0,Y 143.171,Z 285.824,A -85,B 0,C 180,E1 -24330.413,E2 -24330.413} C_VEL
LIN {X 0,Y 144.091,Z 288.37,A -85,B 0,C 180,E1 -24331.418,E2 -24331.418} C_VEL
LIN {X 0,Y 146.142,Z 290.577,A -85,B 0,C 180,E1 -24333.039,E2 -24333.039} C_VEL
LIN {X 0,Y 147.053,Z 291.396,A -85,B 0,C 180,E1 -24333.72,E2 -24333.72} C_VEL
LIN {X 0,Y 148.8,Z 294.569,A -85,B 0,C 180,E1 -24335.247,E2 -24335.247} C_VEL
LIN {X 0,Y 150.25,Z 296.219,A -85,B 0,C 180,E1 -24336.3,E2 -24336.3} C_VEL
LIN {X 0,Y 152.147,Z 299.508,A -85,B 0,C 180,E1 -24337.868,E2 -24337.868} C_VEL
LIN {X 0,Y 156.248,Z 307.471,A -85,B 0,C 180,E1 -24341.311,E2 -24341.311} C_VEL
LIN {X 0,Y 159.781,Z 316.43,A -85,B 0,C 180,E1 -24344.73,E2 -24344.73} C_VEL
LIN {X 0,Y 161.779,Z 324.81,A -85,B 0,C 180,E1 -24347.605,E2 -24347.605} C_VEL
LIN {X 0,Y 162.726,Z 335.269,A -85,B 0,C 180,E1 -24351.024,E2 -24351.024} C_VEL
LIN {X 0,Y 162.393,Z 344.718,A -85,B 0,C 180,E1 -24354.25,E2 -24354.25} C_VEL
LIN {X 0,Y 161.922,Z 346.659,A -85,B 0,C 180,E1 -24354.894,E2 -24354.894} C_VEL
LIN {X 0,Y 157.969,Z 355.485,A -85,B 0,C 180,E1 -24357.732,E2 -24357.732} C_VEL
LIN {X 0,Y 154.498,Z 362.761,A -85,B 0,C 180,E1 -24360.725,E2 -24360.725} C_VEL
LIN {X 0,Y 150.641,Z 369.925,A -85,B 0,C 180,E1 -24364.434,E2 -24364.434} C_VEL
LIN {X 0,Y 147.822,Z 374.755,A -85,B 0,C 180,E1 -24367.645,E2 -24367.645} C_VEL
LIN {X 0,Y 145.187,Z 379.442,A -85,B 0,C 180,E1 -24371.661,E2 -24371.661} C_VEL
LIN {X 0,Y 143.171,Z 383.026,A -85,B 0,C 180,E1 -24375.792,E2 -24375.792} C_VEL
LIN {X 0,Y 142.149,Z 384.876,A -85,B 0,C 180,E1 -24378.594,E2 -24378.594} C_VEL
LIN {X 0,Y 141.435,Z 386.264,A -85,B 0,C 180,E1 -24381.427,E2 -24381.427} C_VEL
LIN {X 0,Y 141.007,Z 387.249,A -85,B 0,C 180,E1 -24384.279,E2 -24384.279} C_VEL
LIN {X 0,Y 140.736,Z 387.855,A -85,B 0,C 180,E1 -24387.138,E2 -24387.138} C_VEL
LIN {X 0,Y 140.69,Z 388.08,A -85,B 0,C 180,E1 -24390,E2 -24390} C_VEL
LIN {X 0,Y 140.737,Z 387.885,A -85,B 0,C 180,E1 -24392.863,E2 -24392.863} C_VEL
LIN {X 0,Y 141.007,Z 387.298,A -85,B 0,C 180,E1 -24395.721,E2 -24395.721} C_VEL
LIN {X 0,Y 142.148,Z 384.975,A -85,B 0,C 180,E1 -24401.407,E2 -24401.407} C_VEL
LIN {X 0,Y 143.751,Z 382.105,A -85,B 0,C 180,E1 -24405.599,E2 -24405.599} C_VEL
LIN {X 0,Y 145.975,Z 378.212,A -85,B 0,C 180,E1 -24409.696,E2 -24409.696} C_VEL
LIN {X 0,Y 148.848,Z 373.187,A -85,B 0,C 180,E1 -24413.662,E2 -24413.662} C_VEL
LIN {X 0,Y 152.44,Z 366.852,A -85,B 0,C 180,E1 -24417.454,E2 -24417.454} C_VEL
LIN {X 0,Y 156.196,Z 359.52,A -85,B 0,C 180,E1 -24420.862,E2 -24420.862} C_VEL
LIN {X 0,Y 160.153,Z 350.86,A -85,B 0,C 180,E1 -24424.021,E2 -24424.021} C_VEL
LIN {X 0,Y 162.458,Z 345.218,A -85,B 0,C 180,E1 -24425.734,E2 -24425.734} C_VEL
LIN {X 0,Y 162.837,Z 335.654,A -85,B 0,C 180,E1 -24429.024,E2 -24429.024} C_VEL
LIN {X 0,Y 162.115,Z 326.992,A -85,B 0,C 180,E1 -24431.894,E2 -24431.894} C_VEL
LIN {X 0,Y 160.636,Z 319.408,A -85,B 0,C 180,E1 -24434.429,E2 -24434.429} C_VEL
LIN {X 0,Y 158.121,Z 311.712,A -85,B 0,C 180,E1 -24437.237,E2 -24437.237} C_VEL
LIN {X 0,Y 154.49,Z 303.853,A -85,B 0,C 180,E1 -24440.44,E2 -24440.44} C_VEL
LIN {X 0,Y 152.235,Z 299.664,A -85,B 0,C 180,E1 -24442.319,E2 -24442.319} C_VEL
LIN {X 0,Y 150.214,Z 296.148,A -85,B 0,C 180,E1 -24444.002,E2 -24444.002} C_VEL
LIN {X 0,Y 147.506,Z 292.542,A -85,B 0,C 180,E1 -24446.106,E2 -24446.106} C_VEL
LIN {X 0,Y 146.77,Z 290.978,A -85,B 0,C 180,E1 -24446.81,E2 -24446.81} C_VEL
LIN {X 0,Y 144.458,Z 288.915,A -85,B 0,C 180,E1 -24448.568,E2 -24448.568} C_VEL
LIN {X 0,Y 143.292,Z 286.509,A -85,B 0,C 180,E1 -24449.717,E2 -24449.717} C_VEL
LIN {X 0,Y 143.137,Z 285.652,A -85,B 0,C 180,E1 -24449.986,E2 -24449.986} C_VEL
LIN {X 0,Y 143.157,Z 285.65,A -85,B 0,C 180,E1 -24453.779,E2 -24453.779} C_VEL
LIN {X 0,Y 143.307,Z 285.632,A -85,B 0,C 180,E1 -24459.922,E2 -24459.922} C_VEL
LIN {X 0,Y 143.326,Z 285.631,A -85,B 0,C 180,E1 -24465.808,E2 -24465.808} C_VEL
LIN {X 0,Y 143.537,Z 285.604,A -85,B 0,C 180,E1 -24468.705,E2 -24468.705} C_VEL
LIN {X 0,Y 143.625,Z 285.594,A -85,B 0,C 180,E1 -24471.558,E2 -24471.558} C_VEL
LIN {X 0,Y 144.159,Z 285.527,A -85,B 0,C 180,E1 -24480,E2 -24480} C_VEL
LIN {X 0,Y 143.628,Z 285.594,A -85,B 0,C 180,E1 -24488.441,E2 -24488.441} C_VEL
LIN {X 0,Y 143.507,Z 285.61,A -85,B 0,C 180,E1 -24491.629,E2 -24491.629} C_VEL
LIN {X 0,Y 143.298,Z 285.633,A -85,B 0,C 180,E1 -24497.114,E2 -24497.114} C_VEL
LIN {X 0,Y 143.276,Z 285.637,A -85,B 0,C 180,E1 -24501.252,E2 -24501.252} C_VEL
LIN {X 0,Y 143.505,Z 287.728,A -85,B 0,C 180,E1 -24508.172,E2 -24508.172} C_VEL
LIN {X 0,Y 143.647,Z 288.601,A -85,B 0,C 180,E1 -24510.301,E2 -24510.301} C_VEL
LIN {X 0,Y 144.981,Z 291.774,A -85,B 0,C 180,E1 -24511.61,E2 -24511.61} C_VEL
LIN {X 0,Y 147.678,Z 295.066,A -85,B 0,C 180,E1 -24513.698,E2 -24513.698} C_VEL
LIN {X 0,Y 149.466,Z 298.742,A -85,B 0,C 180,E1 -24515.273,E2 -24515.273} C_VEL
LIN {X 0,Y 150.856,Z 300.912,A -85,B 0,C 180,E1 -24516.337,E2 -24516.337} C_VEL
LIN {X 0,Y 153.336,Z 305.758,A -85,B 0,C 180,E1 -24518.393,E2 -24518.393} C_VEL
LIN {X 0,Y 156.791,Z 313.489,A -85,B 0,C 180,E1 -24521.388,E2 -24521.388} C_VEL
LIN {X 0,Y 159.672,Z 321.484,A -85,B 0,C 180,E1 -24524.232,E2 -24524.232} C_VEL
LIN {X 0,Y 160.698,Z 325.686,A -85,B 0,C 180,E1 -24525.593,E2 -24525.593} C_VEL
LIN {X 0,Y 161.274,Z 335.349,A -85,B 0,C 180,E1 -24528.344,E2 -24528.344} C_VEL
LIN {X 0,Y 160.903,Z 345.837,A -85,B 0,C 180,E1 -24531.508,E2 -24531.508} C_VEL
LIN {X 0,Y 159.794,Z 354.42,A -85,B 0,C 180,E1 -24534.355,E2 -24534.355} C_VEL
LIN {X 0,Y 158.909,Z 358.183,A -85,B 0,C 180,E1 -24535.675,E2 -24535.675} C_VEL
LIN {X 0,Y 154.285,Z 367.824,A -85,B 0,C 180,E1 -24539.172,E2 -24539.172} C_VEL
LIN {X 0,Y 150.467,Z 375.504,A -85,B 0,C 180,E1 -24542.909,E2 -24542.909} C_VEL
LIN {X 0,Y 146.647,Z 382.59,A -85,B 0,C 180,E1 -24547.455,E2 -24547.455} C_VEL
LIN {X 0,Y 144.025,Z 387.304,A -85,B 0,C 180,E1 -24551.507,E2 -24551.507} C_VEL
LIN {X 0,Y 142.219,Z 390.911,A -85,B 0,C 180,E1 -24555.695,E2 -24555.695} C_VEL
LIN {X 0,Y 141.399,Z 392.773,A -85,B 0,C 180,E1 -24558.532,E2 -24558.532} C_VEL
LIN {X 0,Y 140.848,Z 394.17,A -85,B 0,C 180,E1 -24561.391,E2 -24561.391} C_VEL
LIN {X 0,Y 140.555,Z 395.171,A -85,B 0,C 180,E1 -24564.26,E2 -24564.26} C_VEL
LIN {X 0,Y 140.569,Z 395.969,A -85,B 0,C 180,E1 -24569.356,E2 -24569.356} C_VEL
LIN {X 0,Y 140.486,Z 395.767,A -85,B 0,C 180,E1 -24572.867,E2 -24572.867} C_VEL
LIN {X 0,Y 140.545,Z 395.146,A -85,B 0,C 180,E1 -24575.74,E2 -24575.74} C_VEL
LIN {X 0,Y 140.837,Z 394.136,A -85,B 0,C 180,E1 -24578.61,E2 -24578.61} C_VEL
LIN {X 0,Y 141.397,Z 392.724,A -85,B 0,C 180,E1 -24581.467,E2 -24581.467} C_VEL
LIN {X 0,Y 142.727,Z 389.766,A -85,B 0,C 180,E1 -24585.713,E2 -24585.713} C_VEL
LIN {X 0,Y 144.81,Z 385.773,A -85,B 0,C 180,E1 -24589.86,E2 -24589.86} C_VEL
LIN {X 0,Y 148.154,Z 379.641,A -85,B 0,C 180,E1 -24594.524,E2 -24594.524} C_VEL
LIN {X 0,Y 151.556,Z 373.198,A -85,B 0,C 180,E1 -24598.227,E2 -24598.227} C_VEL
LIN {X 0,Y 155.789,Z 364.648,A -85,B 0,C 180,E1 -24602.01,E2 -24602.01} C_VEL
LIN {X 0,Y 158.871,Z 357.942,A -85,B 0,C 180,E1 -24604.334,E2 -24604.334} C_VEL
LIN {X 0,Y 160.325,Z 350.607,A -85,B 0,C 180,E1 -24606.856,E2 -24606.856} C_VEL
LIN {X 0,Y 161.123,Z 340.524,A -85,B 0,C 180,E1 -24610.043,E2 -24610.043} C_VEL
LIN {X 0,Y 161.008,Z 330.267,A -85,B 0,C 180,E1 -24613.019,E2 -24613.019} C_VEL
LIN {X 0,Y 160.554,Z 325.178,A -85,B 0,C 180,E1 -24614.457,E2 -24614.457} C_VEL
LIN {X 0,Y 158.621,Z 318.437,A -85,B 0,C 180,E1 -24616.713,E2 -24616.713} C_VEL
LIN {X 0,Y 155.251,Z 309.829,A -85,B 0,C 180,E1 -24619.829,E2 -24619.829} C_VEL
LIN {X 0,Y 154.497,Z 308.525,A -85,B 0,C 180,E1 -24620.407,E2 -24620.407} C_VEL
LIN {X 0,Y 152.771,Z 306.643,A -85,B 0,C 180,E1 -24621.557,E2 -24621.557} C_VEL
LIN {X 0,Y 145.769,Z 303.209,A -85,B 0,C 180,E1 -24625.795,E2 -24625.795} C_VEL
LIN {X 0,Y 144.348,Z 301.181,A -85,B 0,C 180,E1 -24627.02,E2 -24627.02} C_VEL
LIN {X 0,Y 143.478,Z 299.794,A -85,B 0,C 180,E1 -24627.812,E2 -24627.812} C_VEL
LIN {X 0,Y 141.291,Z 296.443,A -85,B 0,C 180,E1 -24629.863,E2 -24629.863} C_VEL
LIN {X 0,Y 140.388,Z 294.444,A -85,B 0,C 180,E1 -24630.868,E2 -24630.868} C_VEL
LIN {X 0,Y 137.602,Z 291.237,A -85,B 0,C 180,E1 -24633.557,E2 -24633.557} C_VEL
LIN {X 0,Y 136.422,Z 288.447,A -85,B 0,C 180,E1 -24635.052,E2 -24635.052} C_VEL
LIN {X 0,Y 136.315,Z 288.076,A -85,B 0,C 180,E1 -24635.235,E2 -24635.235} C_VEL
LIN {X 0,Y 136.305,Z 286.985,A -85,B 0,C 180,E1 -24638.843,E2 -24638.843} C_VEL
LIN {X 0,Y 136.242,Z 286.513,A -85,B 0,C 180,E1 -24641.97,E2 -24641.97} C_VEL
LIN {X 0,Y 136.445,Z 286.489,A -85,B 0,C 180,E1 -24648.138,E2 -24648.138} C_VEL
LIN {X 0,Y 136.552,Z 286.475,A -85,B 0,C 180,E1 -24651.118,E2 -24651.118} C_VEL
LIN {X 0,Y 137.125,Z 286.405,A -85,B 0,C 180,E1 -24660,E2 -24660} C_VEL
LIN {X 0,Y 136.55,Z 286.472,A -85,B 0,C 180,E1 -24668.882,E2 -24668.882} C_VEL
LIN {X 0,Y 136.418,Z 286.488,A -85,B 0,C 180,E1 -24671.892,E2 -24671.892} C_VEL
LIN {X 0,Y 136.21,Z 286.515,A -85,B 0,C 180,E1 -24678.034,E2 -24678.034} C_VEL
LIN {X 0,Y 136.197,Z 286.517,A -85,B 0,C 180,E1 -24681.746,E2 -24681.746} C_VEL
LIN {X 0,Y 136.082,Z 286.55,A -85,B 0,C 180,E1 -24684.913,E2 -24684.913} C_VEL
LIN {X 0,Y 136.877,Z 288.957,A -85,B 0,C 180,E1 -24686.081,E2 -24686.081} C_VEL
LIN {X 0,Y 139.007,Z 291.406,A -85,B 0,C 180,E1 -24688.276,E2 -24688.276} C_VEL
LIN {X 0,Y 140.257,Z 292.337,A -85,B 0,C 180,E1 -24689.413,E2 -24689.413} C_VEL
LIN {X 0,Y 141.843,Z 295.435,A -85,B 0,C 180,E1 -24691.142,E2 -24691.142} C_VEL
LIN {X 0,Y 143.796,Z 297.482,A -85,B 0,C 180,E1 -24692.834,E2 -24692.834} C_VEL
LIN {X 0,Y 145.757,Z 300.869,A -85,B 0,C 180,E1 -24694.72,E2 -24694.72} C_VEL
LIN {X 0,Y 146.541,Z 301.901,A -85,B 0,C 180,E1 -24695.383,E2 -24695.383} C_VEL
LIN {X 0,Y 150.035,Z 308.663,A -85,B 0,C 180,E1 -24698.753,E2 -24698.753} C_VEL
LIN {X 0,Y 152.93,Z 315.579,A -85,B 0,C 180,E1 -24701.789,E2 -24701.789} C_VEL
LIN {X 0,Y 155.145,Z 322.61,A -85,B 0,C 180,E1 -24704.6,E2 -24704.6} C_VEL
LIN {X 0,Y 156.251,Z 329.097,A -85,B 0,C 180,E1 -24706.963,E2 -24706.963} C_VEL
LIN {X 0,Y 156.686,Z 338.746,A -85,B 0,C 180,E1 -24710.38,E2 -24710.38} C_VEL
LIN {X 0,Y 156.032,Z 346.867,A -85,B 0,C 180,E1 -24713.358,E2 -24713.358} C_VEL
LIN {X 0,Y 151.887,Z 355.94,A -85,B 0,C 180,E1 -24716.396,E2 -24716.396} C_VEL
LIN {X 0,Y 147.653,Z 364.288,A -85,B 0,C 180,E1 -24720.015,E2 -24720.015} C_VEL
LIN {X 0,Y 143.642,Z 371.151,A -85,B 0,C 180,E1 -24723.874,E2 -24723.874} C_VEL
LIN {X 0,Y 140.288,Z 376.644,A -85,B 0,C 180,E1 -24727.931,E2 -24727.931} C_VEL
LIN {X 0,Y 137.67,Z 380.95,A -85,B 0,C 180,E1 -24732.164,E2 -24732.164} C_VEL
LIN {X 0,Y 136.306,Z 383.226,A -85,B 0,C 180,E1 -24735.061,E2 -24735.061} C_VEL
LIN {X 0,Y 135.185,Z 385.077,A -85,B 0,C 180,E1 -24737.998,E2 -24737.998} C_VEL
LIN {X 0,Y 134.429,Z 386.464,A -85,B 0,C 180,E1 -24740.977,E2 -24740.977} C_VEL
LIN {X 0,Y 133.949,Z 387.449,A -85,B 0,C 180,E1 -24743.977,E2 -24743.977} C_VEL
LIN {X 0,Y 133.579,Z 388.204,A -85,B 0,C 180,E1 -24748.494,E2 -24748.494} C_VEL
LIN {X 0,Y 133.659,Z 388.084,A -85,B 0,C 180,E1 -24753.014,E2 -24753.014} C_VEL
LIN {X 0,Y 133.949,Z 387.498,A -85,B 0,C 180,E1 -24756.024,E2 -24756.024} C_VEL
LIN {X 0,Y 135.183,Z 385.174,A -85,B 0,C 180,E1 -24762.003,E2 -24762.003} C_VEL
LIN {X 0,Y 136.917,Z 382.304,A -85,B 0,C 180,E1 -24766.399,E2 -24766.399} C_VEL
LIN {X 0,Y 139.303,Z 378.41,A -85,B 0,C 180,E1 -24770.681,E2 -24770.681} C_VEL
LIN {X 0,Y 142.364,Z 373.386,A -85,B 0,C 180,E1 -24774.811,E2 -24774.811} C_VEL
LIN {X 0,Y 146.174,Z 367.05,A -85,B 0,C 180,E1 -24778.738,E2 -24778.738} C_VEL
LIN {X 0,Y 149.89,Z 360.212,A -85,B 0,C 180,E1 -24782.048,E2 -24782.048} C_VEL
LIN {X 0,Y 154.333,Z 351.055,A -85,B 0,C 180,E1 -24785.494,E2 -24785.494} C_VEL
LIN {X 0,Y 156.022,Z 347.353,A -85,B 0,C 180,E1 -24786.645,E2 -24786.645} C_VEL
LIN {X 0,Y 156.734,Z 340.126,A -85,B 0,C 180,E1 -24789.318,E2 -24789.318} C_VEL
LIN {X 0,Y 156.52,Z 331.701,A -85,B 0,C 180,E1 -24792.34,E2 -24792.34} C_VEL
LIN {X 0,Y 155.469,Z 324.094,A -85,B 0,C 180,E1 -24795.064,E2 -24795.064} C_VEL
LIN {X 0,Y 153.699,Z 317.643,A -85,B 0,C 180,E1 -24797.588,E2 -24797.588} C_VEL
LIN {X 0,Y 150.606,Z 309.891,A -85,B 0,C 180,E1 -24800.935,E2 -24800.935} C_VEL
LIN {X 0,Y 148.566,Z 305.496,A -85,B 0,C 180,E1 -24802.989,E2 -24802.989} C_VEL
LIN {X 0,Y 146.579,Z 301.914,A -85,B 0,C 180,E1 -24804.875,E2 -24804.875} C_VEL
LIN {X 0,Y 143.854,Z 297.682,A -85,B 0,C 180,E1 -24807.389,E2 -24807.389} C_VEL
LIN {X 0,Y 143.054,Z 296.68,A -85,B 0,C 180,E1 -24808.121,E2 -24808.121} C_VEL
LIN {X 0,Y 140.945,Z 293.978,A -85,B 0,C 180,E1 -24810.09,E2 -24810.09} C_VEL
LIN {X 0,Y 140.174,Z 292.087,A -85,B 0,C 180,E1 -24811.036,E2 -24811.036} C_VEL
LIN {X 0,Y 137.615,Z 290.057,A -85,B 0,C 180,E1 -24813.457,E2 -24813.457} C_VEL
LIN {X 0,Y 136.265,Z 287.508,A -85,B 0,C 180,E1 -24815.123,E2 -24815.123} C_VEL
LIN {X 0,Y 136.083,Z 286.528,A -85,B 0,C 180,E1 -24815.596,E2 -24815.596} C_VEL
LIN {X 0,Y 136.244,Z 286.515,A -85,B 0,C 180,E1 -24818.833,E2 -24818.833} C_VEL
LIN {X 0,Y 136.247,Z 286.511,A -85,B 0,C 180,E1 -24825.053,E2 -24825.053} C_VEL
LIN {X 0,Y 136.427,Z 286.489,A -85,B 0,C 180,E1 -24828.177,E2 -24828.177} C_VEL
LIN {X 0,Y 136.55,Z 286.474,A -85,B 0,C 180,E1 -24831.118,E2 -24831.118} C_VEL
LIN {X 0,Y 137.116,Z 286.404,A -85,B 0,C 180,E1 -24840,E2 -24840} C_VEL
LIN {X 0,Y 136.553,Z 286.476,A -85,B 0,C 180,E1 -24848.882,E2 -24848.882} C_VEL
LIN {X 0,Y 136.442,Z 286.488,A -85,B 0,C 180,E1 -24851.89,E2 -24851.89} C_VEL
LIN {X 0,Y 136.24,Z 286.514,A -85,B 0,C 180,E1 -24858.03,E2 -24858.03} C_VEL
LIN {X 0,Y 136.306,Z 287.256,A -85,B 0,C 180,E1 -24861.86,E2 -24861.86} C_VEL
LIN {X 0,Y 136.354,Z 288.192,A -85,B 0,C 180,E1 -24864.554,E2 -24864.554} C_VEL
LIN {X 0,Y 137.434,Z 290.903,A -85,B 0,C 180,E1 -24865.968,E2 -24865.968} C_VEL
LIN {X 0,Y 139.983,Z 294.053,A -85,B 0,C 180,E1 -24868.529,E2 -24868.529} C_VEL
LIN {X 0,Y 140.788,Z 295.024,A -85,B 0,C 180,E1 -24869.28,E2 -24869.28} C_VEL
LIN {X 0,Y 142.556,Z 298.639,A -85,B 0,C 180,E1 -24871.175,E2 -24871.175} C_VEL
LIN {X 0,Y 144.217,Z 300.811,A -85,B 0,C 180,E1 -24872.622,E2 -24872.622} C_VEL
LIN {X 0,Y 146.302,Z 304.971,A -85,B 0,C 180,E1 -24874.677,E2 -24874.677} C_VEL
LIN {X 0,Y 149.399,Z 311.633,A -85,B 0,C 180,E1 -24877.701,E2 -24877.701} C_VEL
LIN {X 0,Y 151.986,Z 317.895,A -85,B 0,C 180,E1 -24880.344,E2 -24880.344} C_VEL
LIN {X 0,Y 154.754,Z 326.771,A -85,B 0,C 180,E1 -24883.742,E2 -24883.742} C_VEL
LIN {X 0,Y 155.361,Z 332.01,A -85,B 0,C 180,E1 -24885.436,E2 -24885.436} C_VEL
LIN {X 0,Y 155.251,Z 341.976,A -85,B 0,C 180,E1 -24888.543,E2 -24888.543} C_VEL
LIN {X 0,Y 154.229,Z 351.449,A -85,B 0,C 180,E1 -24891.718,E2 -24891.718} C_VEL
LIN {X 0,Y 152.946,Z 357.98,A -85,B 0,C 180,E1 -24894.135,E2 -24894.135} C_VEL
LIN {X 0,Y 148.987,Z 366.139,A -85,B 0,C 180,E1 -24897.147,E2 -24897.147} C_VEL
LIN {X 0,Y 144.716,Z 374.148,A -85,B 0,C 180,E1 -24900.945,E2 -24900.945} C_VEL
LIN {X 0,Y 141.72,Z 379.576,A -85,B 0,C 180,E1 -24904.283,E2 -24904.283} C_VEL
LIN {X 0,Y 138.127,Z 385.67,A -85,B 0,C 180,E1 -24909.135,E2 -24909.135} C_VEL
LIN {X 0,Y 135.868,Z 389.636,A -85,B 0,C 180,E1 -24913.471,E2 -24913.471} C_VEL
LIN {X 0,Y 134.434,Z 392.573,A -85,B 0,C 180,E1 -24917.929,E2 -24917.929} C_VEL
LIN {X 0,Y 133.822,Z 393.971,A -85,B 0,C 180,E1 -24920.935,E2 -24920.935} C_VEL
LIN {X 0,Y 133.398,Z 395.583,A -85,B 0,C 180,E1 -24926.98,E2 -24926.98} C_VEL
LIN {X 0,Y 133.532,Z 395.798,A -85,B 0,C 180,E1 -24930,E2 -24930} C_VEL
LIN {X 0,Y 133.397,Z 395.567,A -85,B 0,C 180,E1 -24933.02,E2 -24933.02} C_VEL
LIN {X 0,Y 133.814,Z 393.936,A -85,B 0,C 180,E1 -24939.065,E2 -24939.065} C_VEL
LIN {X 0,Y 134.432,Z 392.523,A -85,B 0,C 180,E1 -24942.07,E2 -24942.07} C_VEL
LIN {X 0,Y 135.867,Z 389.564,A -85,B 0,C 180,E1 -24946.529,E2 -24946.529} C_VEL
LIN {X 0,Y 138.124,Z 385.572,A -85,B 0,C 180,E1 -24950.865,E2 -24950.865} C_VEL
LIN {X 0,Y 141.718,Z 379.439,A -85,B 0,C 180,E1 -24955.717,E2 -24955.717} C_VEL
LIN {X 0,Y 145.366,Z 372.87,A -85,B 0,C 180,E1 -24959.626,E2 -24959.626} C_VEL
LIN {X 0,Y 149.795,Z 364.445,A -85,B 0,C 180,E1 -24963.455,E2 -24963.455} C_VEL
LIN {X 0,Y 152.236,Z 359.527,A -85,B 0,C 180,E1 -24965.244,E2 -24965.244} C_VEL
LIN {X 0,Y 153.69,Z 354.205,A -85,B 0,C 180,E1 -24967.184,E2 -24967.184} C_VEL
LIN {X 0,Y 154.869,Z 345.286,A -85,B 0,C 180,E1 -24970.291,E2 -24970.291} C_VEL
LIN {X 0,Y 155.299,Z 335.567,A -85,B 0,C 180,E1 -24973.386,E2 -24973.386} C_VEL
LIN {X 0,Y 155.118,Z 328.956,A -85,B 0,C 180,E1 -24975.393,E2 -24975.393} C_VEL
LIN {X 0,Y 153.642,Z 322.936,A -85,B 0,C 180,E1 -24977.569,E2 -24977.569} C_VEL
LIN {X 0,Y 150.197,Z 313.592,A -85,B 0,C 180,E1 -24981.3,E2 -24981.3} C_VEL
LIN {X 0,Y 146.132,Z 304.72,A -85,B 0,C 180,E1 -24985.277,E2 -24985.277} C_VEL
LIN {X 0,Y 144.348,Z 301.181,A -85,B 0,C 180,E1 -24987.02,E2 -24987.02} C_VEL
LIN {X 0,Y 143.137,Z 299.025,A -85,B 0,C 180,E1 -24988.209,E2 -24988.209} C_VEL
LIN {X 0,Y 140.799,Z 296.924,A -85,B 0,C 180,E1 -24990.202,E2 -24990.202} C_VEL
LIN {X 0,Y 136.457,Z 295.191,A -85,B 0,C 180,E1 -24993.854,E2 -24993.854} C_VEL
LIN {X 0,Y 132.582,Z 293.359,A -85,B 0,C 180,E1 -24997.778,E2 -24997.778} C_VEL
LIN {X 0,Y 131.965,Z 292.735,A -85,B 0,C 180,E1 -24998.57,E2 -24998.57} C_VEL
LIN {X 0,Y 129.898,Z 289.714,A -85,B 0,C 180,E1 -25001.773,E2 -25001.773} C_VEL
LIN {X 0,Y 129.196,Z 287.521,A -85,B 0,C 180,E1 -25003.406,E2 -25003.406} C_VEL
LIN {X 0,Y 129.367,Z 287.371,A -85,B 0,C 180,E1 -25007.923,E2 -25007.923} C_VEL
LIN {X 0,Y 129.477,Z 287.357,A -85,B 0,C 180,E1 -25010.628,E2 -25010.628} C_VEL
LIN {X 0,Y 130.08,Z 287.282,A -85,B 0,C 180,E1 -25020,E2 -25020} C_VEL
LIN {X 0,Y 129.472,Z 287.355,A -85,B 0,C 180,E1 -25029.372,E2 -25029.372} C_VEL
LIN {X 0,Y 129.171,Z 287.392,A -85,B 0,C 180,E1 -25035.786,E2 -25035.786} C_VEL
LIN {X 0,Y 129.183,Z 287.572,A -85,B 0,C 180,E1 -25037.309,E2 -25037.309} C_VEL
LIN {X 0,Y 130.122,Z 290.219,A -85,B 0,C 180,E1 -25039.319,E2 -25039.319} C_VEL
LIN {X 0,Y 132.843,Z 292.828,A -85,B 0,C 180,E1 -25043.113,E2 -25043.113} C_VEL
LIN {X 0,Y 133.551,Z 293.359,A -85,B 0,C 180,E1 -25043.966,E2 -25043.966} C_VEL
LIN {X 0,Y 135.004,Z 296.347,A -85,B 0,C 180,E1 -25046.055,E2 -25046.055} C_VEL
LIN {X 0,Y 137.293,Z 298.726,A -85,B 0,C 180,E1 -25048.575,E2 -25048.575} C_VEL
LIN {X 0,Y 138.813,Z 301.582,A -85,B 0,C 180,E1 -25050.418,E2 -25050.418} C_VEL
LIN {X 0,Y 140.042,Z 302.943,A -85,B 0,C 180,E1 -25051.63,E2 -25051.63} C_VEL
LIN {X 0,Y 143.321,Z 308.814,A -85,B 0,C 180,E1 -25055.228,E2 -25055.228} C_VEL
LIN {X 0,Y 146.31,Z 315.319,A -85,B 0,C 180,E1 -25058.642,E2 -25058.642} C_VEL
LIN {X 0,Y 149.109,Z 323.706,A -85,B 0,C 180,E1 -25062.468,E2 -25062.468} C_VEL
LIN {X 0,Y 150.327,Z 330.034,A -85,B 0,C 180,E1 -25065.054,E2 -25065.054} C_VEL
LIN {X 0,Y 150.715,Z 338.405,A -85,B 0,C 180,E1 -25068.254,E2 -25068.254} C_VEL
LIN {X 0,Y 150.313,Z 345.154,A -85,B 0,C 180,E1 -25070.861,E2 -25070.861} C_VEL
LIN {X 0,Y 149.6,Z 349.009,A -85,B 0,C 180,E1 -25072.359,E2 -25072.359} C_VEL
LIN {X 0,Y 144.763,Z 358.537,A -85,B 0,C 180,E1 -25075.822,E2 -25075.822} C_VEL
LIN {X 0,Y 140.064,Z 366.942,A -85,B 0,C 180,E1 -25079.883,E2 -25079.883} C_VEL
LIN {X 0,Y 136.011,Z 373.351,A -85,B 0,C 180,E1 -25083.946,E2 -25083.946} C_VEL
LIN {X 0,Y 132.736,Z 378.428,A -85,B 0,C 180,E1 -25088.246,E2 -25088.246} C_VEL
LIN {X 0,Y 130.141,Z 382.369,A -85,B 0,C 180,E1 -25092.722,E2 -25092.722} C_VEL
LIN {X 0,Y 128.25,Z 385.277,A -85,B 0,C 180,E1 -25097.338,E2 -25097.338} C_VEL
LIN {X 0,Y 127.416,Z 386.664,A -85,B 0,C 180,E1 -25100.476,E2 -25100.476} C_VEL
LIN {X 0,Y 126.888,Z 387.649,A -85,B 0,C 180,E1 -25103.64,E2 -25103.64} C_VEL
LIN {X 0,Y 126.585,Z 388.254,A -85,B 0,C 180,E1 -25106.818,E2 -25106.818} C_VEL
LIN {X 0,Y 126.505,Z 388.479,A -85,B 0,C 180,E1 -25110,E2 -25110} C_VEL
LIN {X 0,Y 126.585,Z 388.283,A -85,B 0,C 180,E1 -25113.183,E2 -25113.183} C_VEL
LIN {X 0,Y 126.889,Z 387.697,A -85,B 0,C 180,E1 -25116.36,E2 -25116.36} C_VEL
LIN {X 0,Y 128.248,Z 385.374,A -85,B 0,C 180,E1 -25122.662,E2 -25122.662} C_VEL
LIN {X 0,Y 130.102,Z 382.504,A -85,B 0,C 180,E1 -25127.284,E2 -25127.284} C_VEL
LIN {X 0,Y 132.682,Z 378.609,A -85,B 0,C 180,E1 -25131.764,E2 -25131.764} C_VEL
LIN {X 0,Y 135.947,Z 373.584,A -85,B 0,C 180,E1 -25136.067,E2 -25136.067} C_VEL
LIN {X 0,Y 139.982,Z 367.248,A -85,B 0,C 180,E1 -25140.137,E2 -25140.137} C_VEL
LIN {X 0,Y 144.698,Z 359.003,A -85,B 0,C 180,E1 -25144.14,E2 -25144.14} C_VEL
LIN {X 0,Y 149.499,Z 349.474,A -85,B 0,C 180,E1 -25147.672,E2 -25147.672} C_VEL
LIN {X 0,Y 150.115,Z 347.559,A -85,B 0,C 180,E1 -25148.341,E2 -25148.341} C_VEL
LIN {X 0,Y 150.777,Z 340.188,A -85,B 0,C 180,E1 -25151.257,E2 -25151.257} C_VEL
LIN {X 0,Y 150.582,Z 331.926,A -85,B 0,C 180,E1 -25154.434,E2 -25154.434} C_VEL
LIN {X 0,Y 149.326,Z 324.276,A -85,B 0,C 180,E1 -25157.497,E2 -25157.497} C_VEL
LIN {X 0,Y 146.893,Z 316.758,A -85,B 0,C 180,E1 -25160.927,E2 -25160.927} C_VEL
LIN {X 0,Y 144.127,Z 310.333,A -85,B 0,C 180,E1 -25164.186,E2 -25164.186} C_VEL
LIN {X 0,Y 140.359,Z 303.42,A -85,B 0,C 180,E1 -25168.345,E2 -25168.345} C_VEL
LIN {X 0,Y 137.775,Z 299.837,A -85,B 0,C 180,E1 -25171.118,E2 -25171.118} C_VEL
LIN {X 0,Y 137.038,Z 298.279,A -85,B 0,C 180,E1 -25172.097,E2 -25172.097} C_VEL
LIN {X 0,Y 134.636,Z 295.776,A -85,B 0,C 180,E1 -25174.801,E2 -25174.801} C_VEL
LIN {X 0,Y 133.36,Z 293.074,A -85,B 0,C 180,E1 -25176.718,E2 -25176.718} C_VEL
LIN {X 0,Y 130.518,Z 290.784,A -85,B 0,C 180,E1 -25180.538,E2 -25180.538} C_VEL
LIN {X 0,Y 129.266,Z 288.013,A -85,B 0,C 180,E1 -25183.008,E2 -25183.008} C_VEL
LIN {X 0,Y 129.149,Z 287.397,A -85,B 0,C 180,E1 -25183.399,E2 -25183.399} C_VEL
LIN {X 0,Y 129.35,Z 287.37,A -85,B 0,C 180,E1 -25187.961,E2 -25187.961} C_VEL
LIN {X 0,Y 129.473,Z 287.355,A -85,B 0,C 180,E1 -25190.628,E2 -25190.628} C_VEL
LIN {X 0,Y 130.072,Z 287.282,A -85,B 0,C 180,E1 -25200,E2 -25200} C_VEL
LIN {X 0,Y 129.476,Z 287.356,A -85,B 0,C 180,E1 -25209.372,E2 -25209.372} C_VEL
LIN {X 0,Y 129.346,Z 287.371,A -85,B 0,C 180,E1 -25212.553,E2 -25212.553} C_VEL
LIN {X 0,Y 129.219,Z 287.601,A -85,B 0,C 180,E1 -25216.286,E2 -25216.286} C_VEL
LIN {X 0,Y 129.763,Z 289.44,A -85,B 0,C 180,E1 -25217.534,E2 -25217.534} C_VEL
LIN {X 0,Y 131.707,Z 292.398,A -85,B 0,C 180,E1 -25220.702,E2 -25220.702} C_VEL
LIN {X 0,Y 133.878,Z 294.707,A -85,B 0,C 180,E1 -25223.493,E2 -25223.493} C_VEL
LIN {X 0,Y 135.742,Z 298.597,A -85,B 0,C 180,E1 -25226.109,E2 -25226.109} C_VEL
LIN {X 0,Y 137.643,Z 300.98,A -85,B 0,C 180,E1 -25228.184,E2 -25228.184} C_VEL
LIN {X 0,Y 139.559,Z 304.901,A -85,B 0,C 180,E1 -25230.507,E2 -25230.507} C_VEL
LIN {X 0,Y 140.229,Z 305.752,A -85,B 0,C 180,E1 -25231.154,E2 -25231.154} C_VEL
LIN {X 0,Y 143.06,Z 311.806,A -85,B 0,C 180,E1 -25234.399,E2 -25234.399} C_VEL
LIN {X 0,Y 146.514,Z 320.644,A -85,B 0,C 180,E1 -25238.578,E2 -25238.578} C_VEL
LIN {X 0,Y 148.947,Z 328.665,A -85,B 0,C 180,E1 -25241.989,E2 -25241.989} C_VEL
LIN {X 0,Y 149.681,Z 333.194,A -85,B 0,C 180,E1 -25243.692,E2 -25243.692} C_VEL
LIN {X 0,Y 149.416,Z 342.242,A -85,B 0,C 180,E1 -25246.706,E2 -25246.706} C_VEL
LIN {X 0,Y 148.35,Z 351.156,A -85,B 0,C 180,E1 -25249.869,E2 -25249.869} C_VEL
LIN {X 0,Y 146.998,Z 357.774,A -85,B 0,C 180,E1 -25252.44,E2 -25252.44} C_VEL
LIN {X 0,Y 145.619,Z 361.243,A -85,B 0,C 180,E1 -25253.756,E2 -25253.756} C_VEL
LIN {X 0,Y 140.64,Z 370.159,A -85,B 0,C 180,E1 -25257.507,E2 -25257.507} C_VEL
LIN {X 0,Y 136.843,Z 377,A -85,B 0,C 180,E1 -25261.374,E2 -25261.374} C_VEL
LIN {X 0,Y 133.55,Z 382.191,A -85,B 0,C 180,E1 -25265.102,E2 -25265.102} C_VEL
LIN {X 0,Y 130.578,Z 386.904,A -85,B 0,C 180,E1 -25269.522,E2 -25269.522} C_VEL
LIN {X 0,Y 128.445,Z 390.511,A -85,B 0,C 180,E1 -25274.122,E2 -25274.122} C_VEL
LIN {X 0,Y 127.463,Z 392.373,A -85,B 0,C 180,E1 -25277.258,E2 -25277.258} C_VEL
LIN {X 0,Y 126.792,Z 393.77,A -85,B 0,C 180,E1 -25280.428,E2 -25280.428} C_VEL
LIN {X 0,Y 126.411,Z 394.771,A -85,B 0,C 180,E1 -25283.616,E2 -25283.616} C_VEL
LIN {X 0,Y 126.303,Z 395.383,A -85,B 0,C 180,E1 -25286.81,E2 -25286.81} C_VEL
LIN {X 0,Y 126.428,Z 395.598,A -85,B 0,C 180,E1 -25290,E2 -25290} C_VEL
LIN {X 0,Y 126.302,Z 395.367,A -85,B 0,C 180,E1 -25293.19,E2 -25293.19} C_VEL
LIN {X 0,Y 126.406,Z 394.745,A -85,B 0,C 180,E1 -25296.384,E2 -25296.384} C_VEL
LIN {X 0,Y 126.785,Z 393.735,A -85,B 0,C 180,E1 -25299.572,E2 -25299.572} C_VEL
LIN {X 0,Y 127.462,Z 392.321,A -85,B 0,C 180,E1 -25302.741,E2 -25302.741} C_VEL
LIN {X 0,Y 129.046,Z 389.363,A -85,B 0,C 180,E1 -25307.43,E2 -25307.43} C_VEL
LIN {X 0,Y 131.491,Z 385.37,A -85,B 0,C 180,E1 -25311.971,E2 -25311.971} C_VEL
LIN {X 0,Y 135.354,Z 379.238,A -85,B 0,C 180,E1 -25317.022,E2 -25317.022} C_VEL
LIN {X 0,Y 139.289,Z 372.543,A -85,B 0,C 180,E1 -25321.143,E2 -25321.143} C_VEL
LIN {X 0,Y 143.913,Z 364.243,A -85,B 0,C 180,E1 -25325.016,E2 -25325.016} C_VEL
LIN {X 0,Y 146.383,Z 359.321,A -85,B 0,C 180,E1 -25326.88,E2 -25326.88} C_VEL
LIN {X 0,Y 147.947,Z 352.841,A -85,B 0,C 180,E1 -25329.399,E2 -25329.399} C_VEL
LIN {X 0,Y 149.22,Z 343.139,A -85,B 0,C 180,E1 -25332.895,E2 -25332.895} C_VEL
LIN {X 0,Y 149.59,Z 334.385,A -85,B 0,C 180,E1 -25335.806,E2 -25335.806} C_VEL
LIN {X 0,Y 149.38,Z 331.011,A -85,B 0,C 180,E1 -25336.961,E2 -25336.961} C_VEL
LIN {X 0,Y 147.571,Z 324.045,A -85,B 0,C 180,E1 -25339.811,E2 -25339.811} C_VEL
LIN {X 0,Y 144.629,Z 315.683,A -85,B 0,C 180,E1 -25343.536,E2 -25343.536} C_VEL
LIN {X 0,Y 141.635,Z 309.027,A -85,B 0,C 180,E1 -25346.919,E2 -25346.919} C_VEL
LIN {X 0,Y 139.912,Z 305.378,A -85,B 0,C 180,E1 -25348.918,E2 -25348.918} C_VEL
LIN {X 0,Y 137.846,Z 301.682,A -85,B 0,C 180,E1 -25351.239,E2 -25351.239} C_VEL
LIN {X 0,Y 137.305,Z 300.453,A -85,B 0,C 180,E1 -25351.949,E2 -25351.949} C_VEL
LIN {X 0,Y 134.758,Z 297.008,A -85,B 0,C 180,E1 -25354.826,E2 -25354.826} C_VEL
LIN {X 0,Y 133.598,Z 294.279,A -85,B 0,C 180,E1 -25356.557,E2 -25356.557} C_VEL
LIN {X 0,Y 131.965,Z 292.735,A -85,B 0,C 180,E1 -25358.57,E2 -25358.57} C_VEL
LIN {X 0,Y 130.165,Z 291.468,A -85,B 0,C 180,E1 -25360.971,E2 -25360.971} C_VEL
LIN {X 0,Y 128.339,Z 291.318,A -85,B 0,C 180,E1 -25363.487,E2 -25363.487} C_VEL
LIN {X 0,Y 124.463,Z 292.206,A -85,B 0,C 180,E1 -25370.571,E2 -25370.571} C_VEL
LIN {X 0,Y 123.921,Z 291.821,A -85,B 0,C 180,E1 -25372.401,E2 -25372.401} C_VEL
LIN {X 0,Y 123.233,Z 289.247,A -85,B 0,C 180,E1 -25380,E2 -25380} C_VEL
LIN {X 0,Y 127.087,Z 294.309,A -85,B 0,C 180,E1 -25396.361,E2 -25396.361} C_VEL
LIN {X 0,Y 128.199,Z 297.14,A -85,B 0,C 180,E1 -25398.996,E2 -25398.996} C_VEL
LIN {X 0,Y 130.874,Z 299.869,A -85,B 0,C 180,E1 -25403.122,E2 -25403.122} C_VEL
LIN {X 0,Y 132.288,Z 302.725,A -85,B 0,C 180,E1 -25405.425,E2 -25405.425} C_VEL
LIN {X 0,Y 134.312,Z 305.47,A -85,B 0,C 180,E1 -25408.095,E2 -25408.095} C_VEL
LIN {X 0,Y 137.036,Z 310.01,A -85,B 0,C 180,E1 -25411.588,E2 -25411.588} C_VEL
LIN {X 0,Y 139.381,Z 314.523,A -85,B 0,C 180,E1 -25414.559,E2 -25414.559} C_VEL
LIN {X 0,Y 141.898,Z 320.816,A -85,B 0,C 180,E1 -25418.071,E2 -25418.071} C_VEL
LIN {X 0,Y 143.963,Z 328.166,A -85,B 0,C 180,E1 -25421.67,E2 -25421.67} C_VEL
LIN {X 0,Y 144.851,Z 335.108,A -85,B 0,C 180,E1 -25424.709,E2 -25424.709} C_VEL
LIN {X 0,Y 144.689,Z 342.667,A -85,B 0,C 180,E1 -25427.821,E2 -25427.821} C_VEL
LIN {X 0,Y 143.858,Z 349.219,A -85,B 0,C 180,E1 -25430.573,E2 -25430.573} C_VEL
LIN {X 0,Y 139.733,Z 357.363,A -85,B 0,C 180,E1 -25433.585,E2 -25433.585} C_VEL
LIN {X 0,Y 134.771,Z 365.918,A -85,B 0,C 180,E1 -25437.689,E2 -25437.689} C_VEL
LIN {X 0,Y 131.034,Z 371.555,A -85,B 0,C 180,E1 -25441.137,E2 -25441.137} C_VEL
LIN {X 0,Y 127.23,Z 377.046,A -85,B 0,C 180,E1 -25445.526,E2 -25445.526} C_VEL
LIN {X 0,Y 124.204,Z 381.352,A -85,B 0,C 180,E1 -25450.153,E2 -25450.153} C_VEL
LIN {X 0,Y 122.616,Z 383.629,A -85,B 0,C 180,E1 -25453.347,E2 -25453.347} C_VEL
LIN {X 0,Y 121.344,Z 385.478,A -85,B 0,C 180,E1 -25456.605,E2 -25456.605} C_VEL
LIN {X 0,Y 120.431,Z 386.864,A -85,B 0,C 180,E1 -25459.918,E2 -25459.918} C_VEL
LIN {X 0,Y 119.84,Z 387.849,A -85,B 0,C 180,E1 -25463.265,E2 -25463.265} C_VEL
LIN {X 0,Y 119.498,Z 388.454,A -85,B 0,C 180,E1 -25466.629,E2 -25466.629} C_VEL
LIN {X 0,Y 119.419,Z 388.678,A -85,B 0,C 180,E1 -25470,E2 -25470} C_VEL
LIN {X 0,Y 119.498,Z 388.483,A -85,B 0,C 180,E1 -25473.372,E2 -25473.372} C_VEL
LIN {X 0,Y 119.841,Z 387.896,A -85,B 0,C 180,E1 -25476.736,E2 -25476.736} C_VEL
LIN {X 0,Y 121.341,Z 385.572,A -85,B 0,C 180,E1 -25483.396,E2 -25483.396} C_VEL
LIN {X 0,Y 123.322,Z 382.703,A -85,B 0,C 180,E1 -25488.267,E2 -25488.267} C_VEL
LIN {X 0,Y 126.094,Z 378.809,A -85,B 0,C 180,E1 -25492.965,E2 -25492.965} C_VEL
LIN {X 0,Y 129.606,Z 373.782,A -85,B 0,C 180,E1 -25497.447,E2 -25497.447} C_VEL
LIN {X 0,Y 133.884,Z 367.446,A -85,B 0,C 180,E1 -25501.664,E2 -25501.664} C_VEL
LIN {X 0,Y 138.613,Z 359.667,A -85,B 0,C 180,E1 -25505.581,E2 -25505.581} C_VEL
LIN {X 0,Y 143,Z 351.449,A -85,B 0,C 180,E1 -25508.802,E2 -25508.802} C_VEL
LIN {X 0,Y 143.834,Z 349.675,A -85,B 0,C 180,E1 -25509.436,E2 -25509.436} C_VEL
LIN {X 0,Y 144.76,Z 342.995,A -85,B 0,C 180,E1 -25512.238,E2 -25512.238} C_VEL
LIN {X 0,Y 144.906,Z 335.612,A -85,B 0,C 180,E1 -25515.313,E2 -25515.313} C_VEL
LIN {X 0,Y 144.205,Z 329.088,A -85,B 0,C 180,E1 -25518.125,E2 -25518.125} C_VEL
LIN {X 0,Y 142.651,Z 322.956,A -85,B 0,C 180,E1 -25521.086,E2 -25521.086} C_VEL
LIN {X 0,Y 140.148,Z 316.049,A -85,B 0,C 180,E1 -25524.782,E2 -25524.782} C_VEL
LIN {X 0,Y 137.864,Z 311.493,A -85,B 0,C 180,E1 -25527.704,E2 -25527.704} C_VEL
LIN {X 0,Y 136.826,Z 309.375,A -85,B 0,C 180,E1 -25529.093,E2 -25529.093} C_VEL
LIN {X 0,Y 134.542,Z 305.865,A -85,B 0,C 180,E1 -25531.957,E2 -25531.957} C_VEL
LIN {X 0,Y 133.952,Z 304.487,A -85,B 0,C 180,E1 -25532.886,E2 -25532.886} C_VEL
LIN {X 0,Y 132.378,Z 302.799,A -85,B 0,C 180,E1 -25534.867,E2 -25534.867} C_VEL
LIN {X 0,Y 130.8,Z 299.595,A -85,B 0,C 180,E1 -25537.49,E2 -25537.49} C_VEL
LIN {X 0,Y 128.166,Z 297.034,A -85,B 0,C 180,E1 -25541.621,E2 -25541.621} C_VEL
LIN {X 0,Y 127.066,Z 294.151,A -85,B 0,C 180,E1 -25544.357,E2 -25544.357} C_VEL
LIN {X 0,Y 123.451,Z 289.888,A -85,B 0,C 180,E1 -25560,E2 -25560} C_VEL
LIN {X 0,Y 127.246,Z 294.408,A -85,B 0,C 180,E1 -25575.312,E2 -25575.312} C_VEL
LIN {X 0,Y 128.836,Z 298.12,A -85,B 0,C 180,E1 -25578.898,E2 -25578.898} C_VEL
LIN {X 0,Y 131.156,Z 300.938,A -85,B 0,C 180,E1 -25582.445,E2 -25582.445} C_VEL
LIN {X 0,Y 132.731,Z 304.525,A -85,B 0,C 180,E1 -25585.062,E2 -25585.062} C_VEL
LIN {X 0,Y 134.418,Z 307.069,A -85,B 0,C 180,E1 -25587.271,E2 -25587.271} C_VEL
LIN {X 0,Y 135.923,Z 310.412,A -85,B 0,C 180,E1 -25589.42,E2 -25589.42} C_VEL
LIN {X 0,Y 137.038,Z 312.551,A -85,B 0,C 180,E1 -25590.854,E2 -25590.854} C_VEL
LIN {X 0,Y 139.624,Z 319.082,A -85,B 0,C 180,E1 -25594.49,E2 -25594.49} C_VEL
LIN {X 0,Y 142.57,Z 328.058,A -85,B 0,C 180,E1 -25598.939,E2 -25598.939} C_VEL
LIN {X 0,Y 143.989,Z 334.706,A -85,B 0,C 180,E1 -25601.899,E2 -25601.899} C_VEL
LIN {X 0,Y 143.811,Z 341.469,A -85,B 0,C 180,E1 -25604.352,E2 -25604.352} C_VEL
LIN {X 0,Y 142.683,Z 350.285,A -85,B 0,C 180,E1 -25607.633,E2 -25607.633} C_VEL
LIN {X 0,Y 140.638,Z 359.369,A -85,B 0,C 180,E1 -25611.343,E2 -25611.343} C_VEL
LIN {X 0,Y 138.111,Z 364.252,A -85,B 0,C 180,E1 -25613.279,E2 -25613.279} C_VEL
LIN {X 0,Y 133.13,Z 372.512,A -85,B 0,C 180,E1 -25617.241,E2 -25617.241} C_VEL
LIN {X 0,Y 129.069,Z 379.179,A -85,B 0,C 180,E1 -25621.546,E2 -25621.546} C_VEL
LIN {X 0,Y 124.919,Z 385.271,A -85,B 0,C 180,E1 -25626.807,E2 -25626.807} C_VEL
LIN {X 0,Y 122.244,Z 389.235,A -85,B 0,C 180,E1 -25631.566,E2 -25631.566} C_VEL
LIN {X 0,Y 120.523,Z 392.173,A -85,B 0,C 180,E1 -25636.511,E2 -25636.511} C_VEL
LIN {X 0,Y 119.784,Z 393.571,A -85,B 0,C 180,E1 -25639.862,E2 -25639.862} C_VEL
LIN {X 0,Y 119.219,Z 395.183,A -85,B 0,C 180,E1 -25646.62,E2 -25646.62} C_VEL
LIN {X 0,Y 119.333,Z 395.399,A -85,B 0,C 180,E1 -25650,E2 -25650} C_VEL
LIN {X 0,Y 119.218,Z 395.167,A -85,B 0,C 180,E1 -25653.379,E2 -25653.379} C_VEL
LIN {X 0,Y 119.756,Z 393.534,A -85,B 0,C 180,E1 -25660.14,E2 -25660.14} C_VEL
LIN {X 0,Y 120.521,Z 392.12,A -85,B 0,C 180,E1 -25663.488,E2 -25663.488} C_VEL
LIN {X 0,Y 122.243,Z 389.161,A -85,B 0,C 180,E1 -25668.433,E2 -25668.433} C_VEL
LIN {X 0,Y 124.915,Z 385.168,A -85,B 0,C 180,E1 -25673.193,E2 -25673.193} C_VEL
LIN {X 0,Y 129.068,Z 379.036,A -85,B 0,C 180,E1 -25678.454,E2 -25678.454} C_VEL
LIN {X 0,Y 133.227,Z 372.34,A -85,B 0,C 180,E1 -25682.732,E2 -25682.732} C_VEL
LIN {X 0,Y 138.133,Z 364.04,A -85,B 0,C 180,E1 -25686.714,E2 -25686.714} C_VEL
LIN {X 0,Y 140.555,Z 359.11,A -85,B 0,C 180,E1 -25688.683,E2 -25688.683} C_VEL
LIN {X 0,Y 142.253,Z 352.011,A -85,B 0,C 180,E1 -25691.602,E2 -25691.602} C_VEL
LIN {X 0,Y 143.636,Z 342.453,A -85,B 0,C 180,E1 -25695.19,E2 -25695.19} C_VEL
LIN {X 0,Y 143.992,Z 335.822,A -85,B 0,C 180,E1 -25697.547,E2 -25697.547} C_VEL
LIN {X 0,Y 143.119,Z 330.647,A -85,B 0,C 180,E1 -25699.749,E2 -25699.749} C_VEL
LIN {X 0,Y 141.019,Z 323.149,A -85,B 0,C 180,E1 -25703.27,E2 -25703.27} C_VEL
LIN {X 0,Y 138.034,Z 315.104,A -85,B 0,C 180,E1 -25707.492,E2 -25707.492} C_VEL
LIN {X 0,Y 136.341,Z 311.143,A -85,B 0,C 180,E1 -25709.829,E2 -25709.829} C_VEL
LIN {X 0,Y 133.89,Z 306.163,A -85,B 0,C 180,E1 -25713.169,E2 -25713.169} C_VEL
LIN {X 0,Y 131.622,Z 302.432,A -85,B 0,C 180,E1 -25716.288,E2 -25716.288} C_VEL
LIN {X 0,Y 130.827,Z 300.478,A -85,B 0,C 180,E1 -25717.704,E2 -25717.704} C_VEL
LIN {X 0,Y 127.873,Z 296.442,A -85,B 0,C 180,E1 -25722.508,E2 -25722.508} C_VEL
LIN {X 0,Y 127.169,Z 294.194,A -85,B 0,C 180,E1 -25724.371,E2 -25724.371} C_VEL
LIN {X 0,Y 123.921,Z 291.821,A -85,B 0,C 180,E1 -25732.401,E2 -25732.401} C_VEL
LIN {X 0,Y 123.448,Z 291.801,A -85,B 0,C 180,E1 -25734.209,E2 -25734.209} C_VEL
LIN {X 0,Y 122.572,Z 293.553,A -85,B 0,C 180,E1 -25737.162,E2 -25737.162} C_VEL
LIN {X 0,Y 121.645,Z 296.671,A -85,B 0,C 180,E1 -25741.375,E2 -25741.375} C_VEL
LIN {X 0,Y 121.616,Z 296.915,A -85,B 0,C 180,E1 -25742.005,E2 -25742.005} C_VEL
LIN {X 0,Y 124.788,Z 301.028,A -85,B 0,C 180,E1 -25755.621,E2 -25755.621} C_VEL
LIN {X 0,Y 125.542,Z 303.26,A -85,B 0,C 180,E1 -25757.884,E2 -25757.884} C_VEL
LIN {X 0,Y 128.078,Z 306.571,A -85,B 0,C 180,E1 -25762.589,E2 -25762.589} C_VEL
LIN {X 0,Y 130.812,Z 311.282,A -85,B 0,C 180,E1 -25767.173,E2 -25767.173} C_VEL
LIN {X 0,Y 133.288,Z 315.872,A -85,B 0,C 180,E1 -25770.937,E2 -25770.937} C_VEL
LIN {X 0,Y 135.738,Z 321.387,A -85,B 0,C 180,E1 -25774.718,E2 -25774.718} C_VEL
LIN {X 0,Y 137.737,Z 328.009,A -85,B 0,C 180,E1 -25778.488,E2 -25778.488} C_VEL
LIN {X 0,Y 138.936,Z 334.325,A -85,B 0,C 180,E1 -25781.746,E2 -25781.746} C_VEL
LIN {X 0,Y 139.068,Z 340.281,A -85,B 0,C 180,E1 -25784.453,E2 -25784.453} C_VEL
LIN {X 0,Y 138.345,Z 347.857,A -85,B 0,C 180,E1 -25787.866,E2 -25787.866} C_VEL
LIN {X 0,Y 137.584,Z 351.218,A -85,B 0,C 180,E1 -25789.361,E2 -25789.361} C_VEL
LIN {X 0,Y 132.678,Z 359.898,A -85,B 0,C 180,E1 -25792.817,E2 -25792.817} C_VEL
LIN {X 0,Y 127.978,Z 367.346,A -85,B 0,C 180,E1 -25796.691,E2 -25796.691} C_VEL
LIN {X 0,Y 123.408,Z 373.754,A -85,B 0,C 180,E1 -25801.049,E2 -25801.049} C_VEL
LIN {X 0,Y 119.623,Z 378.832,A -85,B 0,C 180,E1 -25805.716,E2 -25805.716} C_VEL
LIN {X 0,Y 116.626,Z 382.772,A -85,B 0,C 180,E1 -25810.644,E2 -25810.644} C_VEL
LIN {X 0,Y 114.441,Z 385.678,A -85,B 0,C 180,E1 -25815.78,E2 -25815.78} C_VEL
LIN {X 0,Y 113.435,Z 387.065,A -85,B 0,C 180,E1 -25819.289,E2 -25819.289} C_VEL
LIN {X 0,Y 112.79,Z 388.049,A -85,B 0,C 180,E1 -25822.841,E2 -25822.841} C_VEL
LIN {X 0,Y 112.424,Z 388.653,A -85,B 0,C 180,E1 -25826.416,E2 -25826.416} C_VEL
LIN {X 0,Y 112.335,Z 388.878,A -85,B 0,C 180,E1 -25830,E2 -25830} C_VEL
LIN {X 0,Y 112.424,Z 388.682,A -85,B 0,C 180,E1 -25833.584,E2 -25833.584} C_VEL
LIN {X 0,Y 112.79,Z 388.096,A -85,B 0,C 180,E1 -25837.159,E2 -25837.159} C_VEL
LIN {X 0,Y 114.438,Z 385.772,A -85,B 0,C 180,E1 -25844.221,E2 -25844.221} C_VEL
LIN {X 0,Y 116.587,Z 382.903,A -85,B 0,C 180,E1 -25849.363,E2 -25849.363} C_VEL
LIN {X 0,Y 119.566,Z 379.008,A -85,B 0,C 180,E1 -25854.297,E2 -25854.297} C_VEL
LIN {X 0,Y 123.352,Z 373.981,A -85,B 0,C 180,E1 -25858.966,E2 -25858.966} C_VEL
LIN {X 0,Y 127.89,Z 367.644,A -85,B 0,C 180,E1 -25863.336,E2 -25863.336} C_VEL
LIN {X 0,Y 132.619,Z 360.34,A -85,B 0,C 180,E1 -25867.149,E2 -25867.149} C_VEL
LIN {X 0,Y 137.512,Z 351.647,A -85,B 0,C 180,E1 -25870.665,E2 -25870.665} C_VEL
LIN {X 0,Y 138.373,Z 348.28,A -85,B 0,C 180,E1 -25872.146,E2 -25872.146} C_VEL
LIN {X 0,Y 139.157,Z 340.476,A -85,B 0,C 180,E1 -25875.671,E2 -25875.671} C_VEL
LIN {X 0,Y 139.041,Z 334.773,A -85,B 0,C 180,E1 -25878.272,E2 -25878.272} C_VEL
LIN {X 0,Y 137.999,Z 328.695,A -85,B 0,C 180,E1 -25881.36,E2 -25881.36} C_VEL
LIN {X 0,Y 135.933,Z 321.718,A -85,B 0,C 180,E1 -25885.338,E2 -25885.338} C_VEL
LIN {X 0,Y 133.495,Z 316.223,A -85,B 0,C 180,E1 -25889.116,E2 -25889.116} C_VEL
LIN {X 0,Y 130.825,Z 311.109,A -85,B 0,C 180,E1 -25893.268,E2 -25893.268} C_VEL
LIN {X 0,Y 127.458,Z 305.615,A -85,B 0,C 180,E1 -25898.997,E2 -25898.997} C_VEL
LIN {X 0,Y 125.796,Z 303.68,A -85,B 0,C 180,E1 -25902.103,E2 -25902.103} C_VEL
LIN {X 0,Y 124.708,Z 300.798,A -85,B 0,C 180,E1 -25905.309,E2 -25905.309} C_VEL
LIN {X 0,Y 121.917,Z 296.904,A -85,B 0,C 180,E1 -25920,E2 -25920} C_VEL
LIN {X 0,Y 125.033,Z 301.121,A -85,B 0,C 180,E1 -25934.548,E2 -25934.548} C_VEL
LIN {X 0,Y 126.23,Z 304.292,A -85,B 0,C 180,E1 -25937.831,E2 -25937.831} C_VEL
LIN {X 0,Y 127.977,Z 306.645,A -85,B 0,C 180,E1 -25941,E2 -25941} C_VEL
LIN {X 0,Y 129.483,Z 310.407,A -85,B 0,C 180,E1 -25944.022,E2 -25944.022} C_VEL
LIN {X 0,Y 130.489,Z 311.885,A -85,B 0,C 180,E1 -25945.523,E2 -25945.523} C_VEL
LIN {X 0,Y 133.198,Z 318.351,A -85,B 0,C 180,E1 -25950.083,E2 -25950.083} C_VEL
LIN {X 0,Y 135.347,Z 324.606,A -85,B 0,C 180,E1 -25953.817,E2 -25953.817} C_VEL
LIN {X 0,Y 137.443,Z 332.165,A -85,B 0,C 180,E1 -25957.851,E2 -25957.851} C_VEL
LIN {X 0,Y 138.481,Z 338.147,A -85,B 0,C 180,E1 -25960.753,E2 -25960.753} C_VEL
LIN {X 0,Y 137.759,Z 345.849,A -85,B 0,C 180,E1 -25963.756,E2 -25963.756} C_VEL
LIN {X 0,Y 136.162,Z 354.348,A -85,B 0,C 180,E1 -25967.242,E2 -25967.242} C_VEL
LIN {X 0,Y 134.283,Z 360.843,A -85,B 0,C 180,E1 -25970.123,E2 -25970.123} C_VEL
LIN {X 0,Y 129.737,Z 368.403,A -85,B 0,C 180,E1 -25973.424,E2 -25973.424} C_VEL
LIN {X 0,Y 125.375,Z 375.127,A -85,B 0,C 180,E1 -25977.229,E2 -25977.229} C_VEL
LIN {X 0,Y 122.134,Z 379.972,A -85,B 0,C 180,E1 -25980.717,E2 -25980.717} C_VEL
LIN {X 0,Y 118.41,Z 385.072,A -85,B 0,C 180,E1 -25985.45,E2 -25985.45} C_VEL
LIN {X 0,Y 115.495,Z 389.035,A -85,B 0,C 180,E1 -25990.446,E2 -25990.446} C_VEL
LIN {X 0,Y 113.614,Z 391.973,A -85,B 0,C 180,E1 -25995.674,E2 -25995.674} C_VEL
LIN {X 0,Y 112.776,Z 393.371,A -85,B 0,C 180,E1 -25999.224,E2 -25999.224} C_VEL
LIN {X 0,Y 112.127,Z 394.983,A -85,B 0,C 180,E1 -26006.406,E2 -26006.406} C_VEL
LIN {X 0,Y 112.25,Z 395.199,A -85,B 0,C 180,E1 -26010,E2 -26010} C_VEL
LIN {X 0,Y 112.126,Z 394.967,A -85,B 0,C 180,E1 -26013.593,E2 -26013.593} C_VEL
LIN {X 0,Y 112.754,Z 393.333,A -85,B 0,C 180,E1 -26020.777,E2 -26020.777} C_VEL
LIN {X 0,Y 113.612,Z 391.919,A -85,B 0,C 180,E1 -26024.326,E2 -26024.326} C_VEL
LIN {X 0,Y 115.494,Z 388.959,A -85,B 0,C 180,E1 -26029.553,E2 -26029.553} C_VEL
LIN {X 0,Y 118.406,Z 384.967,A -85,B 0,C 180,E1 -26034.55,E2 -26034.55} C_VEL
LIN {X 0,Y 122.859,Z 378.834,A -85,B 0,C 180,E1 -26040.035,E2 -26040.035} C_VEL
LIN {X 0,Y 127.273,Z 372.136,A -85,B 0,C 180,E1 -26044.472,E2 -26044.472} C_VEL
LIN {X 0,Y 132.5,Z 363.837,A -85,B 0,C 180,E1 -26048.553,E2 -26048.553} C_VEL
LIN {X 0,Y 134.22,Z 360.602,A -85,B 0,C 180,E1 -26049.898,E2 -26049.898} C_VEL
LIN {X 0,Y 136.332,Z 353.041,A -85,B 0,C 180,E1 -26053.209,E2 -26053.209} C_VEL
LIN {X 0,Y 137.895,Z 344.058,A -85,B 0,C 180,E1 -26056.822,E2 -26056.822} C_VEL
LIN {X 0,Y 138.348,Z 337.999,A -85,B 0,C 180,E1 -26059.204,E2 -26059.204} C_VEL
LIN {X 0,Y 137.287,Z 332.035,A -85,B 0,C 180,E1 -26062.099,E2 -26062.099} C_VEL
LIN {X 0,Y 135.113,Z 324.03,A -85,B 0,C 180,E1 -26066.33,E2 -26066.33} C_VEL
LIN {X 0,Y 132.623,Z 316.869,A -85,B 0,C 180,E1 -26070.648,E2 -26070.648} C_VEL
LIN {X 0,Y 130.287,Z 311.689,A -85,B 0,C 180,E1 -26074.435,E2 -26074.435} C_VEL
LIN {X 0,Y 127.699,Z 306.401,A -85,B 0,C 180,E1 -26079.041,E2 -26079.041} C_VEL
LIN {X 0,Y 125.395,Z 302.621,A -85,B 0,C 180,E1 -26083.621,E2 -26083.621} C_VEL
LIN {X 0,Y 124.851,Z 300.873,A -85,B 0,C 180,E1 -26085.327,E2 -26085.327} C_VEL
LIN {X 0,Y 121.722,Z 296.287,A -85,B 0,C 180,E1 -26100,E2 -26100} C_VEL
LIN {X 0,Y 121.616,Z 296.915,A -85,B 0,C 180,E1 -26102.005,E2 -26102.005} C_VEL
LIN {X 0,Y 121.585,Z 298.808,A -85,B 0,C 180,E1 -26105.603,E2 -26105.603} C_VEL
LIN {X 0,Y 121.609,Z 301.752,A -85,B 0,C 180,E1 -26109.057,E2 -26109.057} C_VEL
LIN {X 0,Y 122.4,Z 308.463,A -85,B 0,C 180,E1 -26115.845,E2 -26115.845} C_VEL
LIN {X 0,Y 123.93,Z 311.381,A -85,B 0,C 180,E1 -26119.893,E2 -26119.893} C_VEL
LIN {X 0,Y 124.742,Z 312.459,A -85,B 0,C 180,E1 -26121.482,E2 -26121.482} C_VEL
LIN {X 0,Y 127.102,Z 316.989,A -85,B 0,C 180,E1 -26126.255,E2 -26126.255} C_VEL
LIN {X 0,Y 129.244,Z 321.477,A -85,B 0,C 180,E1 -26130.199,E2 -26130.199} C_VEL
LIN {X 0,Y 131.095,Z 326.192,A -85,B 0,C 180,E1 -26133.705,E2 -26133.705} C_VEL
LIN {X 0,Y 132.565,Z 332.044,A -85,B 0,C 180,E1 -26137.323,E2 -26137.323} C_VEL
LIN {X 0,Y 133.369,Z 336.82,A -85,B 0,C 180,E1 -26140.05,E2 -26140.05} C_VEL
LIN {X 0,Y 133.423,Z 341.643,A -85,B 0,C 180,E1 -26142.486,E2 -26142.486} C_VEL
LIN {X 0,Y 132.652,Z 348.366,A -85,B 0,C 180,E1 -26145.76,E2 -26145.76} C_VEL
LIN {X 0,Y 132.021,Z 351.43,A -85,B 0,C 180,E1 -26147.256,E2 -26147.256} C_VEL
LIN {X 0,Y 130.322,Z 354.877,A -85,B 0,C 180,E1 -26148.653,E2 -26148.653} C_VEL
LIN {X 0,Y 124.706,Z 363.772,A -85,B 0,C 180,E1 -26152.711,E2 -26152.711} C_VEL
LIN {X 0,Y 119.624,Z 370.932,A -85,B 0,C 180,E1 -26157.082,E2 -26157.082} C_VEL
LIN {X 0,Y 115.752,Z 375.762,A -85,B 0,C 180,E1 -26160.94,E2 -26160.94} C_VEL
LIN {X 0,Y 112.022,Z 380.448,A -85,B 0,C 180,E1 -26165.934,E2 -26165.934} C_VEL
LIN {X 0,Y 109.091,Z 384.03,A -85,B 0,C 180,E1 -26171.209,E2 -26171.209} C_VEL
LIN {X 0,Y 107.577,Z 385.879,A -85,B 0,C 180,E1 -26174.852,E2 -26174.852} C_VEL
LIN {X 0,Y 105.745,Z 388.25,A -85,B 0,C 180,E1 -26182.362,E2 -26182.362} C_VEL
LIN {X 0,Y 105.344,Z 388.853,A -85,B 0,C 180,E1 -26186.175,E2 -26186.175} C_VEL
LIN {X 0,Y 105.238,Z 389.078,A -85,B 0,C 180,E1 -26190,E2 -26190} C_VEL
LIN {X 0,Y 105.344,Z 388.882,A -85,B 0,C 180,E1 -26193.826,E2 -26193.826} C_VEL
LIN {X 0,Y 105.745,Z 388.296,A -85,B 0,C 180,E1 -26197.639,E2 -26197.639} C_VEL
LIN {X 0,Y 107.573,Z 385.971,A -85,B 0,C 180,E1 -26205.149,E2 -26205.149} C_VEL
LIN {X 0,Y 109.909,Z 383.102,A -85,B 0,C 180,E1 -26210.591,E2 -26210.591} C_VEL
LIN {X 0,Y 113.112,Z 379.207,A -85,B 0,C 180,E1 -26215.781,E2 -26215.781} C_VEL
LIN {X 0,Y 117.198,Z 374.179,A -85,B 0,C 180,E1 -26220.646,E2 -26220.646} C_VEL
LIN {X 0,Y 122.017,Z 367.842,A -85,B 0,C 180,E1 -26225.169,E2 -26225.169} C_VEL
LIN {X 0,Y 126.727,Z 361.02,A -85,B 0,C 180,E1 -26228.862,E2 -26228.862} C_VEL
LIN {X 0,Y 131.204,Z 353.618,A -85,B 0,C 180,E1 -26232.034,E2 -26232.034} C_VEL
LIN {X 0,Y 132.009,Z 351.851,A -85,B 0,C 180,E1 -26232.75,E2 -26232.75} C_VEL
LIN {X 0,Y 133.103,Z 346.087,A -85,B 0,C 180,E1 -26235.577,E2 -26235.577} C_VEL
LIN {X 0,Y 133.525,Z 338.97,A -85,B 0,C 180,E1 -26239.066,E2 -26239.066} C_VEL
LIN {X 0,Y 133.042,Z 334.219,A -85,B 0,C 180,E1 -26241.647,E2 -26241.647} C_VEL
LIN {X 0,Y 131.786,Z 328.527,A -85,B 0,C 180,E1 -26245.092,E2 -26245.092} C_VEL
LIN {X 0,Y 129.898,Z 322.768,A -85,B 0,C 180,E1 -26249.072,E2 -26249.072} C_VEL
LIN {X 0,Y 127.327,Z 317.294,A -85,B 0,C 180,E1 -26253.796,E2 -26253.796} C_VEL
LIN {X 0,Y 124.966,Z 312.818,A -85,B 0,C 180,E1 -26258.558,E2 -26258.558} C_VEL
LIN {X 0,Y 122.833,Z 309.55,A -85,B 0,C 180,E1 -26263.376,E2 -26263.376} C_VEL
LIN {X 0,Y 122.414,Z 308.16,A -85,B 0,C 180,E1 -26265.027,E2 -26265.027} C_VEL
LIN {X 0,Y 121.886,Z 307.246,A -85,B 0,C 180,E1 -26266.665,E2 -26266.665} C_VEL
LIN {X 0,Y 120.004,Z 303.81,A -85,B 0,C 180,E1 -26280,E2 -26280} C_VEL
LIN {X 0,Y 122.32,Z 307.443,A -85,B 0,C 180,E1 -26293.287,E2 -26293.287} C_VEL
LIN {X 0,Y 123.94,Z 311.399,A -85,B 0,C 180,E1 -26298.172,E2 -26298.172} C_VEL
LIN {X 0,Y 124.703,Z 312.526,A -85,B 0,C 180,E1 -26299.764,E2 -26299.764} C_VEL
LIN {X 0,Y 127.219,Z 318.664,A -85,B 0,C 180,E1 -26305.349,E2 -26305.349} C_VEL
LIN {X 0,Y 129.13,Z 324.017,A -85,B 0,C 180,E1 -26309.33,E2 -26309.33} C_VEL
LIN {X 0,Y 130.864,Z 330.161,A -85,B 0,C 180,E1 -26313.24,E2 -26313.24} C_VEL
LIN {X 0,Y 132.468,Z 337.802,A -85,B 0,C 180,E1 -26317.596,E2 -26317.596} C_VEL
LIN {X 0,Y 132.897,Z 341.205,A -85,B 0,C 180,E1 -26319.39,E2 -26319.39} C_VEL
LIN {X 0,Y 132.159,Z 347.081,A -85,B 0,C 180,E1 -26321.883,E2 -26321.883} C_VEL
LIN {X 0,Y 130.304,Z 355.332,A -85,B 0,C 180,E1 -26325.479,E2 -26325.479} C_VEL
LIN {X 0,Y 128.657,Z 360.636,A -85,B 0,C 180,E1 -26327.997,E2 -26327.997} C_VEL
LIN {X 0,Y 126.977,Z 363.856,A -85,B 0,C 180,E1 -26329.432,E2 -26329.432} C_VEL
LIN {X 0,Y 121.352,Z 372.113,A -85,B 0,C 180,E1 -26333.585,E2 -26333.585} C_VEL
LIN {X 0,Y 116.748,Z 378.782,A -85,B 0,C 180,E1 -26338.214,E2 -26338.214} C_VEL
LIN {X 0,Y 111.974,Z 384.873,A -85,B 0,C 180,E1 -26343.937,E2 -26343.937} C_VEL
LIN {X 0,Y 108.805,Z 388.836,A -85,B 0,C 180,E1 -26349.19,E2 -26349.19} C_VEL
LIN {X 0,Y 106.703,Z 391.772,A -85,B 0,C 180,E1 -26354.724,E2 -26354.724} C_VEL
LIN {X 0,Y 105.796,Z 393.171,A -85,B 0,C 180,E1 -26358.504,E2 -26358.504} C_VEL
LIN {X 0,Y 105.035,Z 394.784,A -85,B 0,C 180,E1 -26366.163,E2 -26366.163} C_VEL
LIN {X 0,Y 105.168,Z 395,A -85,B 0,C 180,E1 -26370,E2 -26370} C_VEL
LIN {X 0,Y 105.035,Z 394.767,A -85,B 0,C 180,E1 -26373.836,E2 -26373.836} C_VEL
LIN {X 0,Y 105.779,Z 393.132,A -85,B 0,C 180,E1 -26381.497,E2 -26381.497} C_VEL
LIN {X 0,Y 106.702,Z 391.717,A -85,B 0,C 180,E1 -26385.275,E2 -26385.275} C_VEL
LIN {X 0,Y 108.804,Z 388.757,A -85,B 0,C 180,E1 -26390.809,E2 -26390.809} C_VEL
LIN {X 0,Y 111.97,Z 384.765,A -85,B 0,C 180,E1 -26396.063,E2 -26396.063} C_VEL
LIN {X 0,Y 116.747,Z 378.632,A -85,B 0,C 180,E1 -26401.785,E2 -26401.785} C_VEL
LIN {X 0,Y 121.437,Z 371.933,A -85,B 0,C 180,E1 -26406.385,E2 -26406.385} C_VEL
LIN {X 0,Y 127.014,Z 363.635,A -85,B 0,C 180,E1 -26410.553,E2 -26410.553} C_VEL
LIN {X 0,Y 128.642,Z 360.391,A -85,B 0,C 180,E1 -26412.009,E2 -26412.009} C_VEL
LIN {X 0,Y 130.942,Z 352.302,A -85,B 0,C 180,E1 -26415.754,E2 -26415.754} C_VEL
LIN {X 0,Y 132.395,Z 344.645,A -85,B 0,C 180,E1 -26419.024,E2 -26419.024} C_VEL
LIN {X 0,Y 132.762,Z 341.059,A -85,B 0,C 180,E1 -26420.562,E2 -26420.562} C_VEL
LIN {X 0,Y 131.768,Z 334.494,A -85,B 0,C 180,E1 -26424.077,E2 -26424.077} C_VEL
LIN {X 0,Y 130.133,Z 327.437,A -85,B 0,C 180,E1 -26428.227,E2 -26428.227} C_VEL
LIN {X 0,Y 128.234,Z 321.523,A -85,B 0,C 180,E1 -26432.233,E2 -26432.233} C_VEL
LIN {X 0,Y 126.689,Z 317.406,A -85,B 0,C 180,E1 -26435.414,E2 -26435.414} C_VEL
LIN {X 0,Y 124.484,Z 312.326,A -85,B 0,C 180,E1 -26440.2,E2 -26440.2} C_VEL
LIN {X 0,Y 123.087,Z 309.895,A -85,B 0,C 180,E1 -26443.412,E2 -26443.412} C_VEL
LIN {X 0,Y 122.597,Z 308.363,A -85,B 0,C 180,E1 -26445.051,E2 -26445.051} C_VEL
LIN {X 0,Y 122.051,Z 307.307,A -85,B 0,C 180,E1 -26446.684,E2 -26446.684} C_VEL
LIN {X 0,Y 119.824,Z 303.249,A -85,B 0,C 180,E1 -26460,E2 -26460} C_VEL
LIN {X 0,Y 122.205,Z 307.711,A -85,B 0,C 180,E1 -26474.999,E2 -26474.999} C_VEL
LIN {X 0,Y 122.4,Z 308.463,A -85,B 0,C 180,E1 -26475.845,E2 -26475.845} C_VEL
LIN {X 0,Y 122.877,Z 311.185,A -85,B 0,C 180,E1 -26478.3,E2 -26478.3} C_VEL
LIN {X 0,Y 123.197,Z 316.899,A -85,B 0,C 180,E1 -26482.086,E2 -26482.086} C_VEL
LIN {X 0,Y 123.844,Z 323.737,A -85,B 0,C 180,E1 -26486.64,E2 -26486.64} C_VEL
LIN {X 0,Y 124.447,Z 325.568,A -85,B 0,C 180,E1 -26488.247,E2 -26488.247} C_VEL
LIN {X 0,Y 126.067,Z 329.982,A -85,B 0,C 180,E1 -26491.981,E2 -26491.981} C_VEL
LIN {X 0,Y 127.186,Z 334.969,A -85,B 0,C 180,E1 -26495.465,E2 -26495.465} C_VEL
LIN {X 0,Y 127.865,Z 340.536,A -85,B 0,C 180,E1 -26498.947,E2 -26498.947} C_VEL
LIN {X 0,Y 127.535,Z 345.983,A -85,B 0,C 180,E1 -26501.892,E2 -26501.892} C_VEL
LIN {X 0,Y 126.481,Z 351.65,A -85,B 0,C 180,E1 -26504.89,E2 -26504.89} C_VEL
LIN {X 0,Y 125.984,Z 353.401,A -85,B 0,C 180,E1 -26505.789,E2 -26505.789} C_VEL
LIN {X 0,Y 121.007,Z 361.291,A -85,B 0,C 180,E1 -26509.235,E2 -26509.235} C_VEL
LIN {X 0,Y 115.478,Z 368.914,A -85,B 0,C 180,E1 -26513.603,E2 -26513.603} C_VEL
LIN {X 0,Y 109.605,Z 375.963,A -85,B 0,C 180,E1 -26519.139,E2 -26519.139} C_VEL
LIN {X 0,Y 105.579,Z 380.649,A -85,B 0,C 180,E1 -26524.363,E2 -26524.363} C_VEL
LIN {X 0,Y 102.374,Z 384.231,A -85,B 0,C 180,E1 -26529.925,E2 -26529.925} C_VEL
LIN {X 0,Y 100.729,Z 386.08,A -85,B 0,C 180,E1 -26533.795,E2 -26533.795} C_VEL
LIN {X 0,Y 99.515,Z 387.465,A -85,B 0,C 180,E1 -26537.769,E2 -26537.769} C_VEL
LIN {X 0,Y 98.704,Z 388.45,A -85,B 0,C 180,E1 -26541.813,E2 -26541.813} C_VEL
LIN {X 0,Y 98.259,Z 389.053,A -85,B 0,C 180,E1 -26545.899,E2 -26545.899} C_VEL
LIN {X 0,Y 98.152,Z 389.277,A -85,B 0,C 180,E1 -26550,E2 -26550} C_VEL
LIN {X 0,Y 98.26,Z 389.081,A -85,B 0,C 180,E1 -26554.102,E2 -26554.102} C_VEL
LIN {X 0,Y 98.704,Z 388.495,A -85,B 0,C 180,E1 -26558.188,E2 -26558.188} C_VEL
LIN {X 0,Y 100.725,Z 386.171,A -85,B 0,C 180,E1 -26566.207,E2 -26566.207} C_VEL
LIN {X 0,Y 103.294,Z 383.301,A -85,B 0,C 180,E1 -26571.976,E2 -26571.976} C_VEL
LIN {X 0,Y 106.745,Z 379.406,A -85,B 0,C 180,E1 -26577.444,E2 -26577.444} C_VEL
LIN {X 0,Y 111.158,Z 374.377,A -85,B 0,C 180,E1 -26582.509,E2 -26582.509} C_VEL
LIN {X 0,Y 116.282,Z 368.04,A -85,B 0,C 180,E1 -26587.186,E2 -26587.186} C_VEL
LIN {X 0,Y 122.16,Z 359.891,A -85,B 0,C 180,E1 -26591.59,E2 -26591.59} C_VEL
LIN {X 0,Y 125.946,Z 353.817,A -85,B 0,C 180,E1 -26594.229,E2 -26594.229} C_VEL
LIN {X 0,Y 127.164,Z 348.958,A -85,B 0,C 180,E1 -26596.752,E2 -26596.752} C_VEL
LIN {X 0,Y 127.942,Z 342.377,A -85,B 0,C 180,E1 -26600.268,E2 -26600.268} C_VEL
LIN {X 0,Y 127.556,Z 336.7,A -85,B 0,C 180,E1 -26603.681,E2 -26603.681} C_VEL
LIN {X 0,Y 126.527,Z 331.488,A -85,B 0,C 180,E1 -26607.209,E2 -26607.209} C_VEL
LIN {X 0,Y 125.138,Z 327.075,A -85,B 0,C 180,E1 -26610.71,E2 -26610.71} C_VEL
LIN {X 0,Y 123.397,Z 322.863,A -85,B 0,C 180,E1 -26614.712,E2 -26614.712} C_VEL
LIN {X 0,Y 121.403,Z 318.566,A -85,B 0,C 180,E1 -26619.675,E2 -26619.675} C_VEL
LIN {X 0,Y 119.661,Z 315.33,A -85,B 0,C 180,E1 -26624.675,E2 -26624.675} C_VEL
LIN {X 0,Y 119.342,Z 314.115,A -85,B 0,C 180,E1 -26626.375,E2 -26626.375} C_VEL
LIN {X 0,Y 117.673,Z 310.57,A -85,B 0,C 180,E1 -26640,E2 -26640} C_VEL
LIN {X 0,Y 118.722,Z 313.298,A -85,B 0,C 180,E1 -26650.229,E2 -26650.229} C_VEL
LIN {X 0,Y 119.767,Z 314.552,A -85,B 0,C 180,E1 -26653.575,E2 -26653.575} C_VEL
LIN {X 0,Y 121.255,Z 318.324,A -85,B 0,C 180,E1 -26658.589,E2 -26658.589} C_VEL
LIN {X 0,Y 123.231,Z 323.924,A -85,B 0,C 180,E1 -26664.146,E2 -26664.146} C_VEL
LIN {X 0,Y 124.854,Z 329.501,A -85,B 0,C 180,E1 -26668.585,E2 -26668.585} C_VEL
LIN {X 0,Y 126.406,Z 336.808,A -85,B 0,C 180,E1 -26673.489,E2 -26673.489} C_VEL
LIN {X 0,Y 127.227,Z 343.292,A -85,B 0,C 180,E1 -26677.419,E2 -26677.419} C_VEL
LIN {X 0,Y 126.97,Z 346.86,A -85,B 0,C 180,E1 -26679.201,E2 -26679.201} C_VEL
LIN {X 0,Y 124.932,Z 355.119,A -85,B 0,C 180,E1 -26683.003,E2 -26683.003} C_VEL
LIN {X 0,Y 122.519,Z 362.075,A -85,B 0,C 180,E1 -26686.5,E2 -26686.5} C_VEL
LIN {X 0,Y 117.62,Z 369.366,A -85,B 0,C 180,E1 -26690.034,E2 -26690.034} C_VEL
LIN {X 0,Y 112.765,Z 375.858,A -85,B 0,C 180,E1 -26694.117,E2 -26694.117} C_VEL
LIN {X 0,Y 108.365,Z 381.394,A -85,B 0,C 180,E1 -26698.745,E2 -26698.745} C_VEL
LIN {X 0,Y 104.366,Z 386.107,A -85,B 0,C 180,E1 -26704.042,E2 -26704.042} C_VEL
LIN {X 0,Y 101.257,Z 389.71,A -85,B 0,C 180,E1 -26709.693,E2 -26709.693} C_VEL
LIN {X 0,Y 99.828,Z 391.572,A -85,B 0,C 180,E1 -26713.644,E2 -26713.644} C_VEL
LIN {X 0,Y 98.811,Z 392.97,A -85,B 0,C 180,E1 -26717.679,E2 -26717.679} C_VEL
LIN {X 0,Y 98.186,Z 393.971,A -85,B 0,C 180,E1 -26721.769,E2 -26721.769} C_VEL
LIN {X 0,Y 97.942,Z 394.584,A -85,B 0,C 180,E1 -26725.885,E2 -26725.885} C_VEL
LIN {X 0,Y 98.074,Z 394.8,A -85,B 0,C 180,E1 -26730,E2 -26730} C_VEL
LIN {X 0,Y 97.941,Z 394.566,A -85,B 0,C 180,E1 -26734.115,E2 -26734.115} C_VEL
LIN {X 0,Y 98.18,Z 393.943,A -85,B 0,C 180,E1 -26738.231,E2 -26738.231} C_VEL
LIN {X 0,Y 98.797,Z 392.931,A -85,B 0,C 180,E1 -26742.322,E2 -26742.322} C_VEL
LIN {X 0,Y 99.827,Z 391.516,A -85,B 0,C 180,E1 -26746.356,E2 -26746.356} C_VEL
LIN {X 0,Y 102.181,Z 388.556,A -85,B 0,C 180,E1 -26752.227,E2 -26752.227} C_VEL
LIN {X 0,Y 105.618,Z 384.564,A -85,B 0,C 180,E1 -26757.761,E2 -26757.761} C_VEL
LIN {X 0,Y 110.738,Z 378.43,A -85,B 0,C 180,E1 -26763.732,E2 -26763.732} C_VEL
LIN {X 0,Y 115.762,Z 371.73,A -85,B 0,C 180,E1 -26768.483,E2 -26768.483} C_VEL
LIN {X 0,Y 121.646,Z 363.43,A -85,B 0,C 180,E1 -26772.753,E2 -26772.753} C_VEL
LIN {X 0,Y 123.127,Z 360.176,A -85,B 0,C 180,E1 -26774.364,E2 -26774.364} C_VEL
LIN {X 0,Y 125.619,Z 352.132,A -85,B 0,C 180,E1 -26778.274,E2 -26778.274} C_VEL
LIN {X 0,Y 127.131,Z 344.96,A -85,B 0,C 180,E1 -26781.544,E2 -26781.544} C_VEL
LIN {X 0,Y 126.774,Z 339.951,A -85,B 0,C 180,E1 -26784.402,E2 -26784.402} C_VEL
LIN {X 0,Y 125.596,Z 332.916,A -85,B 0,C 180,E1 -26788.827,E2 -26788.827} C_VEL
LIN {X 0,Y 124.14,Z 326.996,A -85,B 0,C 180,E1 -26793.07,E2 -26793.07} C_VEL
LIN {X 0,Y 122.863,Z 323.014,A -85,B 0,C 180,E1 -26796.396,E2 -26796.396} C_VEL
LIN {X 0,Y 121.045,Z 318.12,A -85,B 0,C 180,E1 -26801.377,E2 -26801.377} C_VEL
LIN {X 0,Y 119.558,Z 314.277,A -85,B 0,C 180,E1 -26806.401,E2 -26806.401} C_VEL
LIN {X 0,Y 117.535,Z 310.04,A -85,B 0,C 180,E1 -26820,E2 -26820} C_VEL
LIN {X 0,Y 119.103,Z 313.829,A -85,B 0,C 180,E1 -26833.653,E2 -26833.653} C_VEL
LIN {X 0,Y 121.184,Z 318.256,A -85,B 0,C 180,E1 -26840.363,E2 -26840.363} C_VEL
LIN {X 0,Y 123.186,Z 322.568,A -85,B 0,C 180,E1 -26845.334,E2 -26845.334} C_VEL
LIN {X 0,Y 124.447,Z 325.568,A -85,B 0,C 180,E1 -26848.247,E2 -26848.247} C_VEL
LIN {X 0,Y 125.051,Z 327.483,A -85,B 0,C 180,E1 -26849.804,E2 -26849.804} C_VEL
LIN {X 0,Y 125.194,Z 331.141,A -85,B 0,C 180,E1 -26851.94,E2 -26851.94} C_VEL
LIN {X 0,Y 124.63,Z 335.296,A -85,B 0,C 180,E1 -26853.895,E2 -26853.895} C_VEL
LIN {X 0,Y 123.187,Z 341.266,A -85,B 0,C 180,E1 -26856.479,E2 -26856.479} C_VEL
LIN {X 0,Y 122.1,Z 346.695,A -85,B 0,C 180,E1 -26859.283,E2 -26859.283} C_VEL
LIN {X 0,Y 121.104,Z 351.873,A -85,B 0,C 180,E1 -26862.276,E2 -26862.276} C_VEL
LIN {X 0,Y 119.978,Z 355.284,A -85,B 0,C 180,E1 -26864.146,E2 -26864.146} C_VEL
LIN {X 0,Y 113.719,Z 364.177,A -85,B 0,C 180,E1 -26868.367,E2 -26868.367} C_VEL
LIN {X 0,Y 107.965,Z 371.336,A -85,B 0,C 180,E1 -26872.978,E2 -26872.978} C_VEL
LIN {X 0,Y 103.583,Z 376.164,A -85,B 0,C 180,E1 -26877.127,E2 -26877.127} C_VEL
LIN {X 0,Y 99.227,Z 380.85,A -85,B 0,C 180,E1 -26882.589,E2 -26882.589} C_VEL
LIN {X 0,Y 95.728,Z 384.432,A -85,B 0,C 180,E1 -26888.465,E2 -26888.465} C_VEL
LIN {X 0,Y 93.931,Z 386.28,A -85,B 0,C 180,E1 -26892.586,E2 -26892.586} C_VEL
LIN {X 0,Y 92.584,Z 387.666,A -85,B 0,C 180,E1 -26896.837,E2 -26896.837} C_VEL
LIN {X 0,Y 91.693,Z 388.65,A -85,B 0,C 180,E1 -26901.183,E2 -26901.183} C_VEL
LIN {X 0,Y 91.186,Z 389.253,A -85,B 0,C 180,E1 -26905.58,E2 -26905.58} C_VEL
LIN {X 0,Y 91.058,Z 389.477,A -85,B 0,C 180,E1 -26910,E2 -26910} C_VEL
LIN {X 0,Y 91.186,Z 389.281,A -85,B 0,C 180,E1 -26914.421,E2 -26914.421} C_VEL
LIN {X 0,Y 91.693,Z 388.695,A -85,B 0,C 180,E1 -26918.818,E2 -26918.818} C_VEL
LIN {X 0,Y 93.925,Z 386.37,A -85,B 0,C 180,E1 -26927.416,E2 -26927.416} C_VEL
LIN {X 0,Y 96.755,Z 383.499,A -85,B 0,C 180,E1 -26933.548,E2 -26933.548} C_VEL
LIN {X 0,Y 100.482,Z 379.606,A -85,B 0,C 180,E1 -26939.315,E2 -26939.315} C_VEL
LIN {X 0,Y 105.249,Z 374.575,A -85,B 0,C 180,E1 -26944.583,E2 -26944.583} C_VEL
LIN {X 0,Y 110.703,Z 368.238,A -85,B 0,C 180,E1 -26949.41,E2 -26949.41} C_VEL
LIN {X 0,Y 116.512,Z 360.679,A -85,B 0,C 180,E1 -26953.627,E2 -26953.627} C_VEL
LIN {X 0,Y 119.912,Z 355.661,A -85,B 0,C 180,E1 -26955.888,E2 -26955.888} C_VEL
LIN {X 0,Y 121.117,Z 352.28,A -85,B 0,C 180,E1 -26957.718,E2 -26957.718} C_VEL
LIN {X 0,Y 122.311,Z 345.817,A -85,B 0,C 180,E1 -26961.479,E2 -26961.479} C_VEL
LIN {X 0,Y 122.242,Z 340.587,A -85,B 0,C 180,E1 -26964.905,E2 -26964.905} C_VEL
LIN {X 0,Y 121.488,Z 335.645,A -85,B 0,C 180,E1 -26968.624,E2 -26968.624} C_VEL
LIN {X 0,Y 120.417,Z 331.632,A -85,B 0,C 180,E1 -26972.166,E2 -26972.166} C_VEL
LIN {X 0,Y 118.769,Z 327.23,A -85,B 0,C 180,E1 -26976.938,E2 -26976.938} C_VEL
LIN {X 0,Y 117.61,Z 324.207,A -85,B 0,C 180,E1 -26980.812,E2 -26980.812} C_VEL
LIN {X 0,Y 116.278,Z 321.014,A -85,B 0,C 180,E1 -26986.009,E2 -26986.009} C_VEL
LIN {X 0,Y 115.538,Z 319.658,A -85,B 0,C 180,E1 -26989.485,E2 -26989.485} C_VEL
LIN {X 0,Y 114.96,Z 317.2,A -85,B 0,C 180,E1 -27000,E2 -27000} C_VEL
LIN {X 0,Y 115.935,Z 319.941,A -85,B 0,C 180,E1 -27010.478,E2 -27010.478} C_VEL
LIN {X 0,Y 116.737,Z 321.602,A -85,B 0,C 180,E1 -27013.935,E2 -27013.935} C_VEL
LIN {X 0,Y 118.026,Z 325.475,A -85,B 0,C 180,E1 -27019.117,E2 -27019.117} C_VEL
LIN {X 0,Y 119.2,Z 329.672,A -85,B 0,C 180,E1 -27023.452,E2 -27023.452} C_VEL
LIN {X 0,Y 120.376,Z 334.8,A -85,B 0,C 180,E1 -27027.844,E2 -27027.844} C_VEL
LIN {X 0,Y 121.312,Z 341.378,A -85,B 0,C 180,E1 -27032.578,E2 -27032.578} C_VEL
LIN {X 0,Y 121.686,Z 346.62,A -85,B 0,C 180,E1 -27036.043,E2 -27036.043} C_VEL
LIN {X 0,Y 121.256,Z 349.779,A -85,B 0,C 180,E1 -27037.764,E2 -27037.764} C_VEL
LIN {X 0,Y 118.489,Z 358.585,A -85,B 0,C 180,E1 -27042.186,E2 -27042.186} C_VEL
LIN {X 0,Y 116.44,Z 363.456,A -85,B 0,C 180,E1 -27044.83,E2 -27044.83} C_VEL
LIN {X 0,Y 110.209,Z 371.716,A -85,B 0,C 180,E1 -27049.183,E2 -27049.183} C_VEL
LIN {X 0,Y 104.86,Z 378.382,A -85,B 0,C 180,E1 -27054.094,E2 -27054.094} C_VEL
LIN {X 0,Y 99.346,Z 384.473,A -85,B 0,C 180,E1 -27060.317,E2 -27060.317} C_VEL
LIN {X 0,Y 95.61,Z 388.436,A -85,B 0,C 180,E1 -27066.153,E2 -27066.153} C_VEL
LIN {X 0,Y 93.003,Z 391.372,A -85,B 0,C 180,E1 -27072.405,E2 -27072.405} C_VEL
LIN {X 0,Y 91.861,Z 392.77,A -85,B 0,C 180,E1 -27076.731,E2 -27076.731} C_VEL
LIN {X 0,Y 90.871,Z 394.384,A -85,B 0,C 180,E1 -27085.564,E2 -27085.564} C_VEL
LIN {X 0,Y 90.972,Z 394.6,A -85,B 0,C 180,E1 -27090,E2 -27090} C_VEL
LIN {X 0,Y 90.87,Z 394.367,A -85,B 0,C 180,E1 -27094.435,E2 -27094.435} C_VEL
LIN {X 0,Y 91.85,Z 392.73,A -85,B 0,C 180,E1 -27103.27,E2 -27103.27} C_VEL
LIN {X 0,Y 93.002,Z 391.314,A -85,B 0,C 180,E1 -27107.594,E2 -27107.594} C_VEL
LIN {X 0,Y 95.608,Z 388.354,A -85,B 0,C 180,E1 -27113.847,E2 -27113.847} C_VEL
LIN {X 0,Y 99.342,Z 384.361,A -85,B 0,C 180,E1 -27119.684,E2 -27119.684} C_VEL
LIN {X 0,Y 104.88,Z 378.227,A -85,B 0,C 180,E1 -27125.897,E2 -27125.897} C_VEL
LIN {X 0,Y 110.262,Z 371.527,A -85,B 0,C 180,E1 -27130.793,E2 -27130.793} C_VEL
LIN {X 0,Y 116.43,Z 363.224,A -85,B 0,C 180,E1 -27135.174,E2 -27135.174} C_VEL
LIN {X 0,Y 119.237,Z 356.046,A -85,B 0,C 180,E1 -27138.998,E2 -27138.998} C_VEL
LIN {X 0,Y 121.394,Z 348.447,A -85,B 0,C 180,E1 -27142.766,E2 -27142.766} C_VEL
LIN {X 0,Y 121.529,Z 345.253,A -85,B 0,C 180,E1 -27144.669,E2 -27144.669} C_VEL
LIN {X 0,Y 120.996,Z 339.554,A -85,B 0,C 180,E1 -27148.483,E2 -27148.483} C_VEL
LIN {X 0,Y 120.03,Z 333.426,A -85,B 0,C 180,E1 -27153.014,E2 -27153.014} C_VEL
LIN {X 0,Y 118.819,Z 328.479,A -85,B 0,C 180,E1 -27157.389,E2 -27157.389} C_VEL
LIN {X 0,Y 117.884,Z 325.155,A -85,B 0,C 180,E1 -27160.859,E2 -27160.859} C_VEL
LIN {X 0,Y 116.57,Z 321.306,A -85,B 0,C 180,E1 -27166.045,E2 -27166.045} C_VEL
LIN {X 0,Y 115.714,Z 319.716,A -85,B 0,C 180,E1 -27169.502,E2 -27169.502} C_VEL
LIN {X 0,Y 114.843,Z 316.69,A -85,B 0,C 180,E1 -27180,E2 -27180} C_VEL
LIN {X 0,Y 115.295,Z 319.429,A -85,B 0,C 180,E1 -27190.537,E2 -27190.537} C_VEL
LIN {X 0,Y 116.168,Z 321.019,A -85,B 0,C 180,E1 -27194.539,E2 -27194.539} C_VEL
LIN {X 0,Y 117.892,Z 325.213,A -85,B 0,C 180,E1 -27200.958,E2 -27200.958} C_VEL
LIN {X 0,Y 119.614,Z 329.671,A -85,B 0,C 180,E1 -27206.147,E2 -27206.147} C_VEL
LIN {X 0,Y 121.079,Z 333.872,A -85,B 0,C 180,E1 -27210.257,E2 -27210.257} C_VEL
LIN {X 0,Y 121.915,Z 338.496,A -85,B 0,C 180,E1 -27213.859,E2 -27213.859} C_VEL
LIN {X 0,Y 122.303,Z 343.158,A -85,B 0,C 180,E1 -27217.11,E2 -27217.11} C_VEL
LIN {X 0,Y 122.1,Z 346.695,A -85,B 0,C 180,E1 -27219.283,E2 -27219.283} C_VEL
LIN {X 0,Y 121.413,Z 349.294,A -85,B 0,C 180,E1 -27220.61,E2 -27220.61} C_VEL
LIN {X 0,Y 119.979,Z 352.056,A -85,B 0,C 180,E1 -27221.744,E2 -27221.744} C_VEL
LIN {X 0,Y 118.01,Z 354.858,A -85,B 0,C 180,E1 -27222.74,E2 -27222.74} C_VEL
LIN {X 0,Y 113.09,Z 360.307,A -85,B 0,C 180,E1 -27224.545,E2 -27224.545} C_VEL
LIN {X 0,Y 107.891,Z 365.479,A -85,B 0,C 180,E1 -27226.629,E2 -27226.629} C_VEL
LIN {X 0,Y 105.647,Z 367.846,A -85,B 0,C 180,E1 -27227.978,E2 -27227.978} C_VEL
LIN {X 0,Y 99.543,Z 374.558,A -85,B 0,C 180,E1 -27233.122,E2 -27233.122} C_VEL
LIN {X 0,Y 94.398,Z 379.638,A -85,B 0,C 180,E1 -27238.59,E2 -27238.59} C_VEL
LIN {X 0,Y 90.31,Z 383.575,A -85,B 0,C 180,E1 -27244.659,E2 -27244.659} C_VEL
LIN {X 0,Y 87.188,Z 386.48,A -85,B 0,C 180,E1 -27251.191,E2 -27251.191} C_VEL
LIN {X 0,Y 84.68,Z 388.85,A -85,B 0,C 180,E1 -27260.446,E2 -27260.446} C_VEL
LIN {X 0,Y 84.107,Z 389.453,A -85,B 0,C 180,E1 -27265.207,E2 -27265.207} C_VEL
LIN {X 0,Y 83.975,Z 389.676,A -85,B 0,C 180,E1 -27270,E2 -27270} C_VEL
LIN {X 0,Y 84.107,Z 389.48,A -85,B 0,C 180,E1 -27274.794,E2 -27274.794} C_VEL
LIN {X 0,Y 84.68,Z 388.894,A -85,B 0,C 180,E1 -27279.555,E2 -27279.555} C_VEL
LIN {X 0,Y 87.183,Z 386.569,A -85,B 0,C 180,E1 -27288.812,E2 -27288.812} C_VEL
LIN {X 0,Y 90.283,Z 383.699,A -85,B 0,C 180,E1 -27295.35,E2 -27295.35} C_VEL
LIN {X 0,Y 94.344,Z 379.805,A -85,B 0,C 180,E1 -27301.431,E2 -27301.431} C_VEL
LIN {X 0,Y 99.483,Z 374.773,A -85,B 0,C 180,E1 -27306.905,E2 -27306.905} C_VEL
LIN {X 0,Y 105.306,Z 368.436,A -85,B 0,C 180,E1 -27311.867,E2 -27311.867} C_VEL
LIN {X 0,Y 111.888,Z 360.325,A -85,B 0,C 180,E1 -27316.414,E2 -27316.414} C_VEL
LIN {X 0,Y 113.969,Z 357.477,A -85,B 0,C 180,E1 -27317.731,E2 -27317.731} C_VEL
LIN {X 0,Y 114.878,Z 355.867,A -85,B 0,C 180,E1 -27318.542,E2 -27318.542} C_VEL
LIN {X 0,Y 116.346,Z 350.758,A -85,B 0,C 180,E1 -27321.747,E2 -27321.747} C_VEL
LIN {X 0,Y 116.861,Z 347.212,A -85,B 0,C 180,E1 -27324.1,E2 -27324.1} C_VEL
LIN {X 0,Y 116.725,Z 342.085,A -85,B 0,C 180,E1 -27328.077,E2 -27328.077} C_VEL
LIN {X 0,Y 116.261,Z 338.648,A -85,B 0,C 180,E1 -27331.079,E2 -27331.079} C_VEL
LIN {X 0,Y 114.927,Z 333.626,A -85,B 0,C 180,E1 -27336.533,E2 -27336.533} C_VEL
LIN {X 0,Y 113.582,Z 329.739,A -85,B 0,C 180,E1 -27341.978,E2 -27341.978} C_VEL
LIN {X 0,Y 112.856,Z 327.697,A -85,B 0,C 180,E1 -27345.576,E2 -27345.576} C_VEL
LIN {X 0,Y 112.286,Z 326.108,A -85,B 0,C 180,E1 -27349.177,E2 -27349.177} C_VEL
LIN {X 0,Y 111.891,Z 323.667,A -85,B 0,C 180,E1 -27360,E2 -27360} C_VEL
LIN {X 0,Y 112.711,Z 326.486,A -85,B 0,C 180,E1 -27370.781,E2 -27370.781} C_VEL
LIN {X 0,Y 113.603,Z 329.316,A -85,B 0,C 180,E1 -27375.82,E2 -27375.82} C_VEL
LIN {X 0,Y 114.049,Z 330.86,A -85,B 0,C 180,E1 -27377.945,E2 -27377.945} C_VEL
LIN {X 0,Y 114.9,Z 335.059,A -85,B 0,C 180,E1 -27382.602,E2 -27382.602} C_VEL
LIN {X 0,Y 115.656,Z 339.984,A -85,B 0,C 180,E1 -27387.113,E2 -27387.113} C_VEL
LIN {X 0,Y 116.148,Z 347.58,A -85,B 0,C 180,E1 -27392.996,E2 -27392.996} C_VEL
LIN {X 0,Y 115.862,Z 351.606,A -85,B 0,C 180,E1 -27395.689,E2 -27395.689} C_VEL
LIN {X 0,Y 113.215,Z 358.953,A -85,B 0,C 180,E1 -27399.62,E2 -27399.62} C_VEL
LIN {X 0,Y 110.433,Z 364.751,A -85,B 0,C 180,E1 -27402.956,E2 -27402.956} C_VEL
LIN {X 0,Y 103.864,Z 372.753,A -85,B 0,C 180,E1 -27407.417,E2 -27407.417} C_VEL
LIN {X 0,Y 98.276,Z 379.176,A -85,B 0,C 180,E1 -27412.564,E2 -27412.564} C_VEL
LIN {X 0,Y 93.201,Z 384.273,A -85,B 0,C 180,E1 -27418.139,E2 -27418.139} C_VEL
LIN {X 0,Y 89.135,Z 388.236,A -85,B 0,C 180,E1 -27424.3,E2 -27424.3} C_VEL
LIN {X 0,Y 86.236,Z 391.172,A -85,B 0,C 180,E1 -27430.974,E2 -27430.974} C_VEL
LIN {X 0,Y 84.95,Z 392.57,A -85,B 0,C 180,E1 -27435.629,E2 -27435.629} C_VEL
LIN {X 0,Y 84.132,Z 393.572,A -85,B 0,C 180,E1 -27440.382,E2 -27440.382} C_VEL
LIN {X 0,Y 83.787,Z 394.184,A -85,B 0,C 180,E1 -27445.188,E2 -27445.188} C_VEL
LIN {X 0,Y 83.879,Z 394.401,A -85,B 0,C 180,E1 -27450,E2 -27450} C_VEL
LIN {X 0,Y 83.786,Z 394.166,A -85,B 0,C 180,E1 -27454.811,E2 -27454.811} C_VEL
LIN {X 0,Y 84.127,Z 393.542,A -85,B 0,C 180,E1 -27459.618,E2 -27459.618} C_VEL
LIN {X 0,Y 84.941,Z 392.529,A -85,B 0,C 180,E1 -27464.372,E2 -27464.372} C_VEL
LIN {X 0,Y 86.235,Z 391.113,A -85,B 0,C 180,E1 -27469.025,E2 -27469.025} C_VEL
LIN {X 0,Y 89.132,Z 388.153,A -85,B 0,C 180,E1 -27475.7,E2 -27475.7} C_VEL
LIN {X 0,Y 93.197,Z 384.159,A -85,B 0,C 180,E1 -27481.861,E2 -27481.861} C_VEL
LIN {X 0,Y 99.185,Z 378.025,A -85,B 0,C 180,E1 -27488.316,E2 -27488.316} C_VEL
LIN {X 0,Y 104.977,Z 371.325,A -85,B 0,C 180,E1 -27493.331,E2 -27493.331} C_VEL
LIN {X 0,Y 110.421,Z 364.514,A -85,B 0,C 180,E1 -27497.049,E2 -27497.049} C_VEL
LIN {X 0,Y 113.144,Z 358.726,A -85,B 0,C 180,E1 -27500.386,E2 -27500.386} C_VEL
LIN {X 0,Y 115.741,Z 351.391,A -85,B 0,C 180,E1 -27504.313,E2 -27504.313} C_VEL
LIN {X 0,Y 116.007,Z 348.738,A -85,B 0,C 180,E1 -27506.03,E2 -27506.03} C_VEL
LIN {X 0,Y 115.85,Z 343.711,A -85,B 0,C 180,E1 -27509.721,E2 -27509.721} C_VEL
LIN {X 0,Y 115.395,Z 338.628,A -85,B 0,C 180,E1 -27513.797,E2 -27513.797} C_VEL
LIN {X 0,Y 114.562,Z 333.787,A -85,B 0,C 180,E1 -27518.403,E2 -27518.403} C_VEL
LIN {X 0,Y 113.59,Z 329.474,A -85,B 0,C 180,E1 -27523.511,E2 -27523.511} C_VEL
LIN {X 0,Y 113.168,Z 328.089,A -85,B 0,C 180,E1 -27525.617,E2 -27525.617} C_VEL
LIN {X 0,Y 112.518,Z 326.259,A -85,B 0,C 180,E1 -27529.2,E2 -27529.2} C_VEL
LIN {X 0,Y 111.797,Z 323.172,A -85,B 0,C 180,E1 -27540,E2 -27540} C_VEL
LIN {X 0,Y 112.064,Z 325.875,A -85,B 0,C 180,E1 -27550.845,E2 -27550.845} C_VEL
LIN {X 0,Y 112.692,Z 327.353,A -85,B 0,C 180,E1 -27554.446,E2 -27554.446} C_VEL
LIN {X 0,Y 113.806,Z 330.616,A -85,B 0,C 180,E1 -27559.856,E2 -27559.856} C_VEL
LIN {X 0,Y 115.15,Z 334.907,A -85,B 0,C 180,E1 -27565.292,E2 -27565.292} C_VEL
LIN {X 0,Y 116.145,Z 338.31,A -85,B 0,C 180,E1 -27568.953,E2 -27568.953} C_VEL
LIN {X 0,Y 116.694,Z 342.814,A -85,B 0,C 180,E1 -27572.822,E2 -27572.822} C_VEL
LIN {X 0,Y 116.784,Z 346.88,A -85,B 0,C 180,E1 -27575.927,E2 -27575.927} C_VEL
LIN {X 0,Y 116.315,Z 350.337,A -85,B 0,C 180,E1 -27578.235,E2 -27578.235} C_VEL
LIN {X 0,Y 114.862,Z 355.499,A -85,B 0,C 180,E1 -27581.45,E2 -27581.45} C_VEL
LIN {X 0,Y 114.009,Z 357.106,A -85,B 0,C 180,E1 -27582.292,E2 -27582.292} C_VEL
LIN {X 0,Y 107.461,Z 365.703,A -85,B 0,C 180,E1 -27586.631,E2 -27586.631} C_VEL
LIN {X 0,Y 105.647,Z 367.846,A -85,B 0,C 180,E1 -27587.978,E2 -27587.978} C_VEL
LIN {X 0,Y 102.272,Z 371.102,A -85,B 0,C 180,E1 -27589.963,E2 -27589.963} C_VEL
LIN {X 0,Y 95.406,Z 375.912,A -85,B 0,C 180,E1 -27593.045,E2 -27593.045} C_VEL
LIN {X 0,Y 88.704,Z 380.071,A -85,B 0,C 180,E1 -27596.8,E2 -27596.8} C_VEL
LIN {X 0,Y 85.726,Z 382.218,A -85,B 0,C 180,E1 -27599.83,E2 -27599.83} C_VEL
LIN {X 0,Y 82.69,Z 384.833,A -85,B 0,C 180,E1 -27604.852,E2 -27604.852} C_VEL
LIN {X 0,Y 80.486,Z 386.681,A -85,B 0,C 180,E1 -27609.557,E2 -27609.557} C_VEL
LIN {X 0,Y 77.699,Z 389.05,A -85,B 0,C 180,E1 -27619.578,E2 -27619.578} C_VEL
LIN {X 0,Y 77.056,Z 389.653,A -85,B 0,C 180,E1 -27624.767,E2 -27624.767} C_VEL
LIN {X 0,Y 76.896,Z 389.875,A -85,B 0,C 180,E1 -27630.001,E2 -27630.001} C_VEL
LIN {X 0,Y 77.056,Z 389.679,A -85,B 0,C 180,E1 -27635.234,E2 -27635.234} C_VEL
LIN {X 0,Y 77.699,Z 389.093,A -85,B 0,C 180,E1 -27640.423,E2 -27640.423} C_VEL
LIN {X 0,Y 80.479,Z 386.769,A -85,B 0,C 180,E1 -27650.446,E2 -27650.446} C_VEL
LIN {X 0,Y 83.919,Z 383.898,A -85,B 0,C 180,E1 -27657.427,E2 -27657.427} C_VEL
LIN {X 0,Y 88.351,Z 380.004,A -85,B 0,C 180,E1 -27663.837,E2 -27663.837} C_VEL
LIN {X 0,Y 93.892,Z 374.972,A -85,B 0,C 180,E1 -27669.513,E2 -27669.513} C_VEL
LIN {X 0,Y 100.118,Z 368.635,A -85,B 0,C 180,E1 -27674.586,E2 -27674.586} C_VEL
LIN {X 0,Y 106.959,Z 360.712,A -85,B 0,C 180,E1 -27679.079,E2 -27679.079} C_VEL
LIN {X 0,Y 109.209,Z 357.679,A -85,B 0,C 180,E1 -27680.557,E2 -27680.557} C_VEL
LIN {X 0,Y 110.816,Z 352.875,A -85,B 0,C 180,E1 -27683.832,E2 -27683.832} C_VEL
LIN {X 0,Y 111.393,Z 349.623,A -85,B 0,C 180,E1 -27686.285,E2 -27686.285} C_VEL
LIN {X 0,Y 111.431,Z 345.745,A -85,B 0,C 180,E1 -27689.697,E2 -27689.697} C_VEL
LIN {X 0,Y 111.015,Z 341.836,A -85,B 0,C 180,E1 -27693.695,E2 -27693.695} C_VEL
LIN {X 0,Y 110.359,Z 338.736,A -85,B 0,C 180,E1 -27697.536,E2 -27697.536} C_VEL
LIN {X 0,Y 109.364,Z 335.095,A -85,B 0,C 180,E1 -27703.191,E2 -27703.191} C_VEL
LIN {X 0,Y 108.644,Z 332.447,A -85,B 0,C 180,E1 -27708.81,E2 -27708.81} C_VEL
LIN {X 0,Y 108.148,Z 330.657,A -85,B 0,C 180,E1 -27716.274,E2 -27716.274} C_VEL
LIN {X 0,Y 108.468,Z 329.95,A -85,B 0,C 180,E1 -27720,E2 -27720} C_VEL
LIN {X 0,Y 108.576,Z 331.654,A -85,B 0,C 180,E1 -27727.438,E2 -27727.438} C_VEL
LIN {X 0,Y 109.075,Z 332.894,A -85,B 0,C 180,E1 -27731.145,E2 -27731.145} C_VEL
LIN {X 0,Y 109.76,Z 335.729,A -85,B 0,C 180,E1 -27736.164,E2 -27736.164} C_VEL
LIN {X 0,Y 110.273,Z 339.111,A -85,B 0,C 180,E1 -27740.52,E2 -27740.52} C_VEL
LIN {X 0,Y 110.629,Z 343.101,A -85,B 0,C 180,E1 -27744.655,E2 -27744.655} C_VEL
LIN {X 0,Y 110.714,Z 348.583,A -85,B 0,C 180,E1 -27749.469,E2 -27749.469} C_VEL
LIN {X 0,Y 110.524,Z 353.094,A -85,B 0,C 180,E1 -27753.106,E2 -27753.106} C_VEL
LIN {X 0,Y 109.695,Z 355.686,A -85,B 0,C 180,E1 -27754.698,E2 -27754.698} C_VEL
LIN {X 0,Y 106.363,Z 363.037,A -85,B 0,C 180,E1 -27759.068,E2 -27759.068} C_VEL
LIN {X 0,Y 104.528,Z 366.04,A -85,B 0,C 180,E1 -27760.852,E2 -27760.852} C_VEL
LIN {X 0,Y 97.557,Z 373.82,A -85,B 0,C 180,E1 -27765.525,E2 -27765.525} C_VEL
LIN {X 0,Y 90.807,Z 380.798,A -85,B 0,C 180,E1 -27771.745,E2 -27771.745} C_VEL
LIN {X 0,Y 85.647,Z 385.508,A -85,B 0,C 180,E1 -27777.765,E2 -27777.765} C_VEL
LIN {X 0,Y 81.511,Z 389.11,A -85,B 0,C 180,E1 -27784.461,E2 -27784.461} C_VEL
LIN {X 0,Y 79.519,Z 390.971,A -85,B 0,C 180,E1 -27789.296,E2 -27789.296} C_VEL
LIN {X 0,Y 78.055,Z 392.37,A -85,B 0,C 180,E1 -27794.328,E2 -27794.328} C_VEL
LIN {X 0,Y 77.12,Z 393.371,A -85,B 0,C 180,E1 -27799.498,E2 -27799.498} C_VEL
LIN {X 0,Y 76.707,Z 393.985,A -85,B 0,C 180,E1 -27804.743,E2 -27804.743} C_VEL
LIN {X 0,Y 76.777,Z 394.201,A -85,B 0,C 180,E1 -27809.999,E2 -27809.999} C_VEL
LIN {X 0,Y 76.706,Z 393.966,A -85,B 0,C 180,E1 -27815.256,E2 -27815.256} C_VEL
LIN {X 0,Y 77.115,Z 393.341,A -85,B 0,C 180,E1 -27820.502,E2 -27820.502} C_VEL
LIN {X 0,Y 78.048,Z 392.328,A -85,B 0,C 180,E1 -27825.672,E2 -27825.672} C_VEL
LIN {X 0,Y 79.518,Z 390.911,A -85,B 0,C 180,E1 -27830.703,E2 -27830.703} C_VEL
LIN {X 0,Y 82.768,Z 387.951,A -85,B 0,C 180,E1 -27837.841,E2 -27837.841} C_VEL
LIN {X 0,Y 87.21,Z 383.957,A -85,B 0,C 180,E1 -27844.34,E2 -27844.34} C_VEL
LIN {X 0,Y 93.667,Z 377.822,A -85,B 0,C 180,E1 -27851.035,E2 -27851.035} C_VEL
LIN {X 0,Y 99.907,Z 371.122,A -85,B 0,C 180,E1 -27856.14,E2 -27856.14} C_VEL
LIN {X 0,Y 104.534,Z 365.804,A -85,B 0,C 180,E1 -27859.144,E2 -27859.144} C_VEL
LIN {X 0,Y 106.35,Z 362.795,A -85,B 0,C 180,E1 -27860.939,E2 -27860.939} C_VEL
LIN {X 0,Y 109.657,Z 355.415,A -85,B 0,C 180,E1 -27865.309,E2 -27865.309} C_VEL
LIN {X 0,Y 110.409,Z 352.765,A -85,B 0,C 180,E1 -27866.984,E2 -27866.984} C_VEL
LIN {X 0,Y 110.615,Z 347.123,A -85,B 0,C 180,E1 -27871.544,E2 -27871.544} C_VEL
LIN {X 0,Y 110.499,Z 342.564,A -85,B 0,C 180,E1 -27875.602,E2 -27875.602} C_VEL
LIN {X 0,Y 110.105,Z 338.921,A -85,B 0,C 180,E1 -27879.448,E2 -27879.448} C_VEL
LIN {X 0,Y 109.583,Z 335.219,A -85,B 0,C 180,E1 -27884.156,E2 -27884.156} C_VEL
LIN {X 0,Y 108.898,Z 332.665,A -85,B 0,C 180,E1 -27888.836,E2 -27888.836} C_VEL
LIN {X 0,Y 108.174,Z 330.46,A -85,B 0,C 180,E1 -27896.275,E2 -27896.275} C_VEL
LIN {X 0,Y 108.394,Z 329.487,A -85,B 0,C 180,E1 -27900,E2 -27900} C_VEL
LIN {X 0,Y 108.45,Z 332.192,A -85,B 0,C 180,E1 -27911.211,E2 -27911.211} C_VEL
LIN {X 0,Y 109.184,Z 334.837,A -85,B 0,C 180,E1 -27916.838,E2 -27916.838} C_VEL
LIN {X 0,Y 110.182,Z 338.491,A -85,B 0,C 180,E1 -27922.502,E2 -27922.502} C_VEL
LIN {X 0,Y 111.126,Z 342.745,A -85,B 0,C 180,E1 -27927.699,E2 -27927.699} C_VEL
LIN {X 0,Y 111.386,Z 346.708,A -85,B 0,C 180,E1 -27931.495,E2 -27931.495} C_VEL
LIN {X 0,Y 111.1,Z 351.176,A -85,B 0,C 180,E1 -27935.2,E2 -27935.2} C_VEL
LIN {X 0,Y 109.777,Z 355.81,A -85,B 0,C 180,E1 -27938.429,E2 -27938.429} C_VEL
LIN {X 0,Y 109.197,Z 357.316,A -85,B 0,C 180,E1 -27939.437,E2 -27939.437} C_VEL
LIN {X 0,Y 105.949,Z 361.671,A -85,B 0,C 180,E1 -27941.556,E2 -27941.556} C_VEL
LIN {X 0,Y 99.145,Z 369.518,A -85,B 0,C 180,E1 -27946.28,E2 -27946.28} C_VEL
LIN {X 0,Y 92.005,Z 376.566,A -85,B 0,C 180,E1 -27952.332,E2 -27952.332} C_VEL
LIN {X 0,Y 86.833,Z 381.253,A -85,B 0,C 180,E1 -27958.259,E2 -27958.259} C_VEL
LIN {X 0,Y 85.726,Z 382.218,A -85,B 0,C 180,E1 -27959.83,E2 -27959.83} C_VEL
LIN {X 0,Y 82.96,Z 384.164,A -85,B 0,C 180,E1 -27963.12,E2 -27963.12} C_VEL
LIN {X 0,Y 77.254,Z 386.816,A -85,B 0,C 180,E1 -27968.605,E2 -27968.605} C_VEL
LIN {X 0,Y 73.013,Z 388.368,A -85,B 0,C 180,E1 -27973.615,E2 -27973.615} C_VEL
LIN {X 0,Y 70.904,Z 389.169,A -85,B 0,C 180,E1 -27977.985,E2 -27977.985} C_VEL
LIN {X 0,Y 70.538,Z 389.359,A -85,B 0,C 180,E1 -27979.552,E2 -27979.552} C_VEL
LIN {X 0,Y 69.815,Z 390.075,A -85,B 0,C 180,E1 -27990.001,E2 -27990.001} C_VEL
LIN {X 0,Y 70,Z 389.879,A -85,B 0,C 180,E1 -27995.763,E2 -27995.763} C_VEL
LIN {X 0,Y 72.009,Z 388.326,A -85,B 0,C 180,E1 -28007.026,E2 -28007.026} C_VEL
LIN {X 0,Y 73.861,Z 386.968,A -85,B 0,C 180,E1 -28012.372,E2 -28012.372} C_VEL
LIN {X 0,Y 77.67,Z 384.097,A -85,B 0,C 180,E1 -28019.847,E2 -28019.847} C_VEL
LIN {X 0,Y 82.537,Z 380.203,A -85,B 0,C 180,E1 -28026.588,E2 -28026.588} C_VEL
LIN {X 0,Y 88.526,Z 375.171,A -85,B 0,C 180,E1 -28032.44,E2 -28032.44} C_VEL
LIN {X 0,Y 95.182,Z 368.833,A -85,B 0,C 180,E1 -28037.594,E2 -28037.594} C_VEL
LIN {X 0,Y 102.446,Z 360.91,A -85,B 0,C 180,E1 -28042.083,E2 -28042.083} C_VEL
LIN {X 0,Y 103.64,Z 359.432,A -85,B 0,C 180,E1 -28042.824,E2 -28042.824} C_VEL
LIN {X 0,Y 105.222,Z 355.586,A -85,B 0,C 180,E1 -28045.676,E2 -28045.676} C_VEL
LIN {X 0,Y 105.875,Z 352.875,A -85,B 0,C 180,E1 -28047.924,E2 -28047.924} C_VEL
LIN {X 0,Y 106.125,Z 348.447,A -85,B 0,C 180,E1 -28052.382,E2 -28052.382} C_VEL
LIN {X 0,Y 105.775,Z 345.161,A -85,B 0,C 180,E1 -28056.505,E2 -28056.505} C_VEL
LIN {X 0,Y 105.388,Z 342.442,A -85,B 0,C 180,E1 -28060.522,E2 -28060.522} C_VEL
LIN {X 0,Y 104.95,Z 340.288,A -85,B 0,C 180,E1 -28064.463,E2 -28064.463} C_VEL
LIN {X 0,Y 104.639,Z 338.614,A -85,B 0,C 180,E1 -28068.376,E2 -28068.376} C_VEL
LIN {X 0,Y 104.355,Z 337.47,A -85,B 0,C 180,E1 -28072.259,E2 -28072.259} C_VEL
LIN {X 0,Y 104.669,Z 335.999,A -85,B 0,C 180,E1 -28080,E2 -28080} C_VEL
LIN {X 0,Y 104.704,Z 337.728,A -85,B 0,C 180,E1 -28087.715,E2 -28087.715} C_VEL
LIN {X 0,Y 105.267,Z 340.074,A -85,B 0,C 180,E1 -28093.513,E2 -28093.513} C_VEL
LIN {X 0,Y 105.4,Z 342.23,A -85,B 0,C 180,E1 -28096.853,E2 -28096.853} C_VEL
LIN {X 0,Y 105.605,Z 344.074,A -85,B 0,C 180,E1 -28099.436,E2 -28099.436} C_VEL
LIN {X 0,Y 105.594,Z 348.736,A -85,B 0,C 180,E1 -28104.581,E2 -28104.581} C_VEL
LIN {X 0,Y 105.188,Z 354.201,A -85,B 0,C 180,E1 -28109.705,E2 -28109.705} C_VEL
LIN {X 0,Y 104.706,Z 356.865,A -85,B 0,C 180,E1 -28111.962,E2 -28111.962} C_VEL
LIN {X 0,Y 100.832,Z 364.335,A -85,B 0,C 180,E1 -28116.721,E2 -28116.721} C_VEL
LIN {X 0,Y 99.917,Z 365.837,A -85,B 0,C 180,E1 -28117.692,E2 -28117.692} C_VEL
LIN {X 0,Y 92.723,Z 373.509,A -85,B 0,C 180,E1 -28122.352,E2 -28122.352} C_VEL
LIN {X 0,Y 85.33,Z 380.599,A -85,B 0,C 180,E1 -28128.783,E2 -28128.783} C_VEL
LIN {X 0,Y 79.707,Z 385.309,A -85,B 0,C 180,E1 -28135.031,E2 -28135.031} C_VEL
LIN {X 0,Y 75.138,Z 388.91,A -85,B 0,C 180,E1 -28142.116,E2 -28142.116} C_VEL
LIN {X 0,Y 72.891,Z 390.771,A -85,B 0,C 180,E1 -28147.314,E2 -28147.314} C_VEL
LIN {X 0,Y 70.141,Z 393.172,A -85,B 0,C 180,E1 -28158.439,E2 -28158.439} C_VEL
LIN {X 0,Y 69.621,Z 393.784,A -85,B 0,C 180,E1 -28164.206,E2 -28164.206} C_VEL
LIN {X 0,Y 69.697,Z 394.002,A -85,B 0,C 180,E1 -28169.999,E2 -28169.999} C_VEL
LIN {X 0,Y 69.619,Z 393.766,A -85,B 0,C 180,E1 -28175.793,E2 -28175.793} C_VEL
LIN {X 0,Y 70.137,Z 393.141,A -85,B 0,C 180,E1 -28181.56,E2 -28181.56} C_VEL
LIN {X 0,Y 71.212,Z 392.127,A -85,B 0,C 180,E1 -28187.221,E2 -28187.221} C_VEL
LIN {X 0,Y 72.89,Z 390.71,A -85,B 0,C 180,E1 -28192.685,E2 -28192.685} C_VEL
LIN {X 0,Y 76.541,Z 387.75,A -85,B 0,C 180,E1 -28200.331,E2 -28200.331} C_VEL
LIN {X 0,Y 81.416,Z 383.755,A -85,B 0,C 180,E1 -28207.175,E2 -28207.175} C_VEL
LIN {X 0,Y 87.311,Z 378.681,A -85,B 0,C 180,E1 -28213.077,E2 -28213.077} C_VEL
LIN {X 0,Y 93.92,Z 372.157,A -85,B 0,C 180,E1 -28218.442,E2 -28218.442} C_VEL
LIN {X 0,Y 99.906,Z 365.596,A -85,B 0,C 180,E1 -28222.316,E2 -28222.316} C_VEL
LIN {X 0,Y 104.125,Z 357.796,A -85,B 0,C 180,E1 -28227.319,E2 -28227.319} C_VEL
LIN {X 0,Y 104.858,Z 355.497,A -85,B 0,C 180,E1 -28228.964,E2 -28228.964} C_VEL
LIN {X 0,Y 105.32,Z 351.226,A -85,B 0,C 180,E1 -28232.781,E2 -28232.781} C_VEL
LIN {X 0,Y 105.501,Z 346.357,A -85,B 0,C 180,E1 -28237.662,E2 -28237.662} C_VEL
LIN {X 0,Y 105.32,Z 342.803,A -85,B 0,C 180,E1 -28242.01,E2 -28242.01} C_VEL
LIN {X 0,Y 105.305,Z 340.923,A -85,B 0,C 180,E1 -28244.517,E2 -28244.517} C_VEL
LIN {X 0,Y 104.91,Z 338.897,A -85,B 0,C 180,E1 -28248.406,E2 -28248.406} C_VEL
LIN {X 0,Y 104.537,Z 337.494,A -85,B 0,C 180,E1 -28252.273,E2 -28252.273} C_VEL
LIN {X 0,Y 104.61,Z 335.588,A -85,B 0,C 180,E1 -28260,E2 -28260} C_VEL
LIN {X 0,Y 104.178,Z 337.219,A -85,B 0,C 180,E1 -28267.754,E2 -28267.754} C_VEL
LIN {X 0,Y 104.477,Z 338.337,A -85,B 0,C 180,E1 -28271.643,E2 -28271.643} C_VEL
LIN {X 0,Y 104.999,Z 341.028,A -85,B 0,C 180,E1 -28277.53,E2 -28277.53} C_VEL
LIN {X 0,Y 105.646,Z 344.876,A -85,B 0,C 180,E1 -28283.525,E2 -28283.525} C_VEL
LIN {X 0,Y 106.057,Z 348.112,A -85,B 0,C 180,E1 -28287.637,E2 -28287.637} C_VEL
LIN {X 0,Y 105.777,Z 352.603,A -85,B 0,C 180,E1 -28292.109,E2 -28292.109} C_VEL
